        g_0:=[[starting_x + 1.5 * scaling, starting_y + 1 * scaling, starting_z + 20],[0,0,1,0],[0,0,0,0],[9E+09,9E+09,9E+09,9E+09,9E+09,9E+09]];
        g_1:=[[starting_x + 1.5 * scaling, starting_y + 1 * scaling, starting_z + 0],[0,0,1,0],[0,0,0,0],[9E+09,9E+09,9E+09,9E+09,9E+09,9E+09]];
        g_2:=[[starting_x + 0 * scaling, starting_y - 1 * scaling, starting_z + 0],[0,0,1,0],[0,0,0,0],[9E+09,9E+09,9E+09,9E+09,9E+09,9E+09]];
        g_3:=[[starting_x + 1 * scaling, starting_y - 3 * scaling, starting_z + 0],[0,0,1,0],[0,0,0,0],[9E+09,9E+09,9E+09,9E+09,9E+09,9E+09]];
        g_4:=[[starting_x + 3.5 * scaling, starting_y - 3.5 * scaling, starting_z + 0],[0,0,1,0],[0,0,0,0],[9E+09,9E+09,9E+09,9E+09,9E+09,9E+09]];
        g_5:=[[starting_x + 6 * scaling, starting_y - 2.5 * scaling, starting_z + 0],[0,0,1,0],[0,0,0,0],[9E+09,9E+09,9E+09,9E+09,9E+09,9E+09]];
        g_6:=[[starting_x + 7 * scaling, starting_y - 1 * scaling, starting_z + 0],[0,0,1,0],[0,0,0,0],[9E+09,9E+09,9E+09,9E+09,9E+09,9E+09]];
        g_7:=[[starting_x + 6 * scaling, starting_y + 1 * scaling, starting_z + 0],[0,0,1,0],[0,0,0,0],[9E+09,9E+09,9E+09,9E+09,9E+09,9E+09]];
        g_8:=[[starting_x + 1.5 * scaling, starting_y + 1 * scaling, starting_z + 0],[0,0,1,0],[0,0,0,0],[9E+09,9E+09,9E+09,9E+09,9E+09,9E+09]];
        g_9:=[[starting_x + 0 * scaling, starting_y + 2.5 * scaling, starting_z + 0],[0,0,1,0],[0,0,0,0],[9E+09,9E+09,9E+09,9E+09,9E+09,9E+09]];
        g_10:=[[starting_x + 1 * scaling, starting_y + 4 * scaling, starting_z + 0],[0,0,1,0],[0,0,0,0],[9E+09,9E+09,9E+09,9E+09,9E+09,9E+09]];
        g_11:=[[starting_x + 0 * scaling, starting_y + 6.5 * scaling, starting_z + 0],[0,0,1,0],[0,0,0,0],[9E+09,9E+09,9E+09,9E+09,9E+09,9E+09]];
        g_12:=[[starting_x + 3 * scaling, starting_y + 9 * scaling, starting_z + 0],[0,0,1,0],[0,0,0,0],[9E+09,9E+09,9E+09,9E+09,9E+09,9E+09]];
        g_13:=[[starting_x + 7.5 * scaling, starting_y + 9 * scaling, starting_z + 0],[0,0,1,0],[0,0,0,0],[9E+09,9E+09,9E+09,9E+09,9E+09,9E+09]];
        g_14:=[[starting_x + 4 * scaling, starting_y + 9 * scaling, starting_z + 0],[0,0,1,0],[0,0,0,0],[9E+09,9E+09,9E+09,9E+09,9E+09,9E+09]];
        g_15:=[[starting_x + 6 * scaling, starting_y + 7 * scaling, starting_z + 0],[0,0,1,0],[0,0,0,0],[9E+09,9E+09,9E+09,9E+09,9E+09,9E+09]];
        g_16:=[[starting_x + 6 * scaling, starting_y + 5 * scaling, starting_z + 0],[0,0,1,0],[0,0,0,0],[9E+09,9E+09,9E+09,9E+09,9E+09,9E+09]];
        g_17:=[[starting_x + 3.5 * scaling, starting_y + 3.5 * scaling, starting_z + 0],[0,0,1,0],[0,0,0,0],[9E+09,9E+09,9E+09,9E+09,9E+09,9E+09]];
        g_18:=[[starting_x + 1 * scaling, starting_y + 4 * scaling, starting_z + 0],[0,0,1,0],[0,0,0,0],[9E+09,9E+09,9E+09,9E+09,9E+09,9E+09]];
        g_19:=[[starting_x + 1 * scaling, starting_y + 4 * scaling, starting_z + 20],[0,0,1,0],[0,0,0,0],[9E+09,9E+09,9E+09,9E+09,9E+09,9E+09]];


        MoveL g_0,v50,fine,MyNewTool\WObj:=A3;
        MoveL g_1,v50,fine,MyNewTool\WObj:=A3;
	    MoveC g_2,g_3,v50,z1,MyNewTool\WObj:=A3;
        MoveC g_4,g_5,v50,z5,MyNewTool\WObj:=A3;
        MoveC g_6,g_7,v50,z5,MyNewTool\WObj:=A3;
        MoveL g_8,v50,fine,MyNewTool\WObj:=A3;
        MoveC g_9,g_10,v50,fine,MyNewTool\WObj:=A3;
        MoveC g_11,g_12,v50,fine,MyNewTool\WObj:=A3;
	    MoveL g_13,v50,fine,MyNewTool\WObj:=A3;
        MoveL g_14,v50,fine,MyNewTool\WObj:=A3;
        MoveC g_15,g_16,v50,z1,MyNewTool\WObj:=A3;
        MoveC g_17,g_18,v50,fine,MyNewTool\WObj:=A3;
        MoveL g_19,v50,fine,MyNewTool\WObj:=A3;


    ENDPROC


    PROC h(num starting_x, num starting_y, num starting_z, num scaling)
        VAR robtarget h_0;
        VAR robtarget h_1;
        VAR robtarget h_2;
	    VAR robtarget h_3;
	    VAR robtarget h_4;
	    VAR robtarget h_5;
	    VAR robtarget h_6;
        VAR robtarget h_7;
        VAR robtarget h_8;
        VAR robtarget h_9;

        h_0:=[[starting_x + 0 * scaling, starting_y + 0 * scaling, starting_z + 20],[0,0,1,0],[0,0,0,0],[9E+09,9E+09,9E+09,9E+09,9E+09,9E+09]];
        h_1:=[[starting_x + 0 * scaling, starting_y + 0 * scaling, starting_z + 0],[0,0,1,0],[0,0,0,0],[9E+09,9E+09,9E+09,9E+09,9E+09,9E+09]];
        h_2:=[[starting_x + 0 * scaling, starting_y + 14 * scaling, starting_z + 0],[0,0,1,0],[0,0,0,0],[9E+09,9E+09,9E+09,9E+09,9E+09,9E+09]];
        h_3:=[[starting_x + 0 * scaling, starting_y + 7 * scaling, starting_z + 0],[0,0,1,0],[0,0,0,0],[9E+09,9E+09,9E+09,9E+09,9E+09,9E+09]];
        h_4:=[[starting_x + 2 * scaling, starting_y + 8 * scaling, starting_z + 0],[0,0,1,0],[0,0,0,0],[9E+09,9E+09,9E+09,9E+09,9E+09,9E+09]];
        h_5:=[[starting_x + 4 * scaling, starting_y + 9 * scaling, starting_z + 0],[0,0,1,0],[0,0,0,0],[9E+09,9E+09,9E+09,9E+09,9E+09,9E+09]];
        h_6:=[[starting_x + 5.8 * scaling, starting_y + 7.2 * scaling, starting_z + 0],[0,0,1,0],[0,0,0,0],[9E+09,9E+09,9E+09,9E+09,9E+09,9E+09]];
        h_7:=[[starting_x + 6 * scaling, starting_y + 6 * scaling, starting_z + 0],[0,0,1,0],[0,0,0,0],[9E+09,9E+09,9E+09,9E+09,9E+09,9E+09]];
        h_8:=[[starting_x + 6 * scaling, starting_y + 0 * scaling, starting_z + 0],[0,0,1,0],[0,0,0,0],[9E+09,9E+09,9E+09,9E+09,9E+09,9E+09]];
        h_9:=[[starting_x + 6 * scaling, starting_y + 0 * scaling, starting_z + 20],[0,0,1,0],[0,0,0,0],[9E+09,9E+09,9E+09,9E+09,9E+09,9E+09]];

        MoveL h_0,v50,fine,MyNewTool\WObj:=A3;
        MoveL h_1,v50,fine,MyNewTool\WObj:=A3;
        MoveL h_2,v50,fine,MyNewTool\WObj:=A3;
        MoveL h_3,v50,fine,MyNewTool\WObj:=A3;
	    MoveL h_4,v50,fine,MyNewTool\WObj:=A3;
        MoveL h_5,v50,z5,MyNewTool\WObj:=A3;
        MoveC h_6,h_7,v50,fine,MyNewTool\WObj:=A3;
        MoveL h_8,v50,fine,MyNewTool\WObj:=A3;
        MoveL h_9,v50,fine,MyNewTool\WObj:=A3;

    ENDPROC

    PROC i(num starting_x, num starting_y, num starting_z, num scaling)
        VAR robtarget i_0;
        VAR robtarget i_1;
        VAR robtarget i_2;
	    VAR robtarget i_3;
	    VAR robtarget i_4;
	    VAR robtarget i_5;
	    VAR robtarget i_6;
        VAR robtarget i_7;


        i_0:=[[starting_x + 0 * scaling, starting_y + 0 * scaling, starting_z + 20],[0,0,1,0],[0,0,0,0],[9E+09,9E+09,9E+09,9E+09,9E+09,9E+09]];
        i_1:=[[starting_x + 0 * scaling, starting_y + 0 * scaling, starting_z + 0],[0,0,1,0],[0,0,0,0],[9E+09,9E+09,9E+09,9E+09,9E+09,9E+09]];
        i_2:=[[starting_x + 0 * scaling, starting_y + 9.5 * scaling, starting_z + 0],[0,0,1,0],[0,0,0,0],[9E+09,9E+09,9E+09,9E+09,9E+09,9E+09]];
        i_3:=[[starting_x + 0 * scaling, starting_y + 9.5 * scaling, starting_z + 20],[0,0,1,0],[0,0,0,0],[9E+09,9E+09,9E+09,9E+09,9E+09,9E+09]];
        i_4:=[[starting_x + 0 * scaling, starting_y + 12 * scaling, starting_z + 20],[0,0,1,0],[0,0,0,0],[9E+09,9E+09,9E+09,9E+09,9E+09,9E+09]];
        i_5:=[[starting_x + 0 * scaling, starting_y + 12 * scaling, starting_z + 0],[0,0,1,0],[0,0,0,0],[9E+09,9E+09,9E+09,9E+09,9E+09,9E+09]];
        i_6:=[[starting_x + 0 * scaling, starting_y + 12.1 * scaling, starting_z + 0],[0,0,1,0],[0,0,0,0],[9E+09,9E+09,9E+09,9E+09,9E+09,9E+09]];
        i_7:=[[starting_x + 0 * scaling, starting_y + 12.1 * scaling, starting_z + 20],[0,0,1,0],[0,0,0,0],[9E+09,9E+09,9E+09,9E+09,9E+09,9E+09]];


        MoveL i_0,v50,fine,MyNewTool\WObj:=A3;
        MoveL i_1,v50,fine,MyNewTool\WObj:=A3;
        MoveL i_2,v50,fine,MyNewTool\WObj:=A3;
        MoveL i_3,v50,fine,MyNewTool\WObj:=A3;
	    MoveL i_4,v50,fine,MyNewTool\WObj:=A3;
        MoveL i_5,v50,fine,MyNewTool\WObj:=A3;
        MoveL i_6,v50,fine,MyNewTool\WObj:=A3;
        MoveL i_7,v50,fine,MyNewTool\WObj:=A3;

    ENDPROC

    PROC j(num starting_x, num starting_y, num starting_z, num scaling)
        VAR robtarget j_0;
        VAR robtarget j_1;
        VAR robtarget j_2;
	    VAR robtarget j_3;
	    VAR robtarget j_4;
	    VAR robtarget j_5;
	    VAR robtarget j_6;
        VAR robtarget j_7;
        VAR robtarget j_8;
        VAR robtarget j_9;

        j_0:=[[starting_x - 1 * scaling, starting_y - 3 * scaling, starting_z + 20],[0,0,1,0],[0,0,0,0],[9E+09,9E+09,9E+09,9E+09,9E+09,9E+09]];
        j_1:=[[starting_x - 1 * scaling, starting_y - 3 * scaling, starting_z + 0],[0,0,1,0],[0,0,0,0],[9E+09,9E+09,9E+09,9E+09,9E+09,9E+09]];
        j_2:=[[starting_x + 1 * scaling, starting_y - 2.5 * scaling, starting_z + 0],[0,0,1,0],[0,0,0,0],[9E+09,9E+09,9E+09,9E+09,9E+09,9E+09]];
        j_3:=[[starting_x + 2 * scaling, starting_y - 1 * scaling, starting_z + 0],[0,0,1,0],[0,0,0,0],[9E+09,9E+09,9E+09,9E+09,9E+09,9E+09]];
        j_4:=[[starting_x + 2 * scaling, starting_y + 9.5 * scaling, starting_z + 0],[0,0,1,0],[0,0,0,0],[9E+09,9E+09,9E+09,9E+09,9E+09,9E+09]];
        j_5:=[[starting_x + 2 * scaling, starting_y + 9.5 * scaling, starting_z + 20],[0,0,1,0],[0,0,0,0],[9E+09,9E+09,9E+09,9E+09,9E+09,9E+09]];
        j_6:=[[starting_x + 2 * scaling, starting_y + 12 * scaling, starting_z + 20],[0,0,1,0],[0,0,0,0],[9E+09,9E+09,9E+09,9E+09,9E+09,9E+09]];
        j_7:=[[starting_x + 2 * scaling, starting_y + 12 * scaling, starting_z + 0],[0,0,1,0],[0,0,0,0],[9E+09,9E+09,9E+09,9E+09,9E+09,9E+09]];
        j_8:=[[starting_x + 2 * scaling, starting_y + 12.1 * scaling, starting_z + 0],[0,0,1,0],[0,0,0,0],[9E+09,9E+09,9E+09,9E+09,9E+09,9E+09]];
        j_9:=[[starting_x + 2 * scaling, starting_y + 12.1 * scaling, starting_z + 20],[0,0,1,0],[0,0,0,0],[9E+09,9E+09,9E+09,9E+09,9E+09,9E+09]];

        MoveL j_0,v50,fine,MyNewTool\WObj:=A3;
        MoveL j_1,v50,fine,MyNewTool\WObj:=A3;
        MoveC j_2,j_3,v50,z1,MyNewTool\WObj:=A3;
        MoveL j_4,v50,fine,MyNewTool\WObj:=A3;
	    MoveL j_5,v50,fine,MyNewTool\WObj:=A3;
        MoveL j_6,v50,fine,MyNewTool\WObj:=A3;
        MoveL j_7,v50,fine,MyNewTool\WObj:=A3;
        MoveL j_8,v50,fine,MyNewTool\WObj:=A3;
        MoveL j_9,v50,fine,MyNewTool\WObj:=A3;

    ENDPROC

    PROC k(num starting_x, num starting_y, num starting_z, num scaling)
        VAR robtarget k_0;
        VAR robtarget k_1;
        VAR robtarget k_2;
	    VAR robtarget k_3;
	    VAR robtarget k_4;
	    VAR robtarget k_5;
	    VAR robtarget k_6;
        VAR robtarget k_7;

        k_0:=[[starting_x + 0 * scaling, starting_y + 14 * scaling, starting_z + 20],[0,0,1,0],[0,0,0,0],[9E+09,9E+09,9E+09,9E+09,9E+09,9E+09]];
        k_1:=[[starting_x + 0 * scaling, starting_y + 14 * scaling, starting_z + 0],[0,0,1,0],[0,0,0,0],[9E+09,9E+09,9E+09,9E+09,9E+09,9E+09]];
        k_2:=[[starting_x + 0 * scaling, starting_y + 0 * scaling, starting_z + 0],[0,0,1,0],[0,0,0,0],[9E+09,9E+09,9E+09,9E+09,9E+09,9E+09]];
        k_3:=[[starting_x + 0 * scaling, starting_y + 5 * scaling, starting_z + 0],[0,0,1,0],[0,0,0,0],[9E+09,9E+09,9E+09,9E+09,9E+09,9E+09]];
        k_4:=[[starting_x + 5.8 * scaling, starting_y + 9 * scaling, starting_z + 0],[0,0,1,0],[0,0,0,0],[9E+09,9E+09,9E+09,9E+09,9E+09,9E+09]];
        k_5:=[[starting_x + 0 * scaling, starting_y + 5 * scaling, starting_z + 0],[0,0,1,0],[0,0,0,0],[9E+09,9E+09,9E+09,9E+09,9E+09,9E+09]];
        k_6:=[[starting_x + 6.2 * scaling, starting_y + 0 * scaling, starting_z + 0],[0,0,1,0],[0,0,0,0],[9E+09,9E+09,9E+09,9E+09,9E+09,9E+09]];
        k_7:=[[starting_x + 6.2 * scaling, starting_y + 0 * scaling, starting_z + 20],[0,0,1,0],[0,0,0,0],[9E+09,9E+09,9E+09,9E+09,9E+09,9E+09]];


        MoveL k_0,v50,fine,MyNewTool\WObj:=A3;
        MoveL k_1,v50,fine,MyNewTool\WObj:=A3;
        MoveL k_2,v50,fine,MyNewTool\WObj:=A3;
        MoveL k_3,v50,fine,MyNewTool\WObj:=A3;
	    MoveL k_4,v50,fine,MyNewTool\WObj:=A3;
        MoveL k_5,v50,z5,MyNewTool\WObj:=A3;
        MoveL k_6,v50,fine,MyNewTool\WObj:=A3;
        MoveL k_7,v50,fine,MyNewTool\WObj:=A3;

    ENDPROC
    PROC l(num starting_x, num starting_y, num starting_z, num scaling)
        VAR robtarget l_0;
        VAR robtarget l_1;
        VAR robtarget l_2;
        VAR robtarget l_3;


        l_0:=[[starting_x + 0 * scaling, starting_y + 0 * scaling, starting_z + 20],[0,0,1,0],[0,0,0,0],[9E+09,9E+09,9E+09,9E+09,9E+09,9E+09]];
        l_1:=[[starting_x + 0 * scaling, starting_y + 0 * scaling, starting_z + 0],[0,0,1,0],[0,0,0,0],[9E+09,9E+09,9E+09,9E+09,9E+09,9E+09]];
        l_2:=[[starting_x + 0 * scaling, starting_y + 14 * scaling, starting_z + 0],[0,0,1,0],[0,0,0,0],[9E+09,9E+09,9E+09,9E+09,9E+09,9E+09]];
        l_3:=[[starting_x + 0 * scaling, starting_y + 14 * scaling, starting_z + 20],[0,0,1,0],[0,0,0,0],[9E+09,9E+09,9E+09,9E+09,9E+09,9E+09]];


        MoveL l_0,v50,fine,MyNewTool\WObj:=A3;
        MoveL l_1,v50,fine,MyNewTool\WObj:=A3;
        MoveL l_2,v50,fine,MyNewTool\WObj:=A3;
        MoveL l_3,v50,fine,MyNewTool\WObj:=A3;

    ENDPROC

    PROC m(num starting_x, num starting_y, num starting_z, num scaling)
        VAR robtarget m_0;
        VAR robtarget m_1;
        VAR robtarget m_2;
        VAR robtarget m_3;
        VAR robtarget m_4;
        VAR robtarget m_5;
        VAR robtarget m_6;
        VAR robtarget m_7;
        VAR robtarget m_8;
        VAR robtarget m_9;
        VAR robtarget m_10;
        VAR robtarget m_11;
        VAR robtarget m_12;
        VAR robtarget m_13;


        m_0:=[[starting_x + 0 * scaling, starting_y + 0 * scaling, starting_z + 20],[0,0,1,0],[0,0,0,0],[9E+09,9E+09,9E+09,9E+09,9E+09,9E+09]];
        m_1:=[[starting_x + 0 * scaling, starting_y + 0 * scaling, starting_z + 0],[0,0,1,0],[0,0,0,0],[9E+09,9E+09,9E+09,9E+09,9E+09,9E+09]];
        m_2:=[[starting_x + 0 * scaling, starting_y + 9.5 * scaling, starting_z + 0],[0,0,1,0],[0,0,0,0],[9E+09,9E+09,9E+09,9E+09,9E+09,9E+09]];
        m_3:=[[starting_x + 0 * scaling, starting_y + 7 * scaling, starting_z + 0],[0,0,1,0],[0,0,0,0],[9E+09,9E+09,9E+09,9E+09,9E+09,9E+09]];
        m_4:=[[starting_x + 2 * scaling, starting_y + 8.5 * scaling, starting_z + 0],[0,0,1,0],[0,0,0,0],[9E+09,9E+09,9E+09,9E+09,9E+09,9E+09]];
        m_5:=[[starting_x + 4 * scaling, starting_y + 9 * scaling, starting_z + 0],[0,0,1,0],[0,0,0,0],[9E+09,9E+09,9E+09,9E+09,9E+09,9E+09]];
        m_6:=[[starting_x + 6 * scaling, starting_y + 8 * scaling, starting_z + 0],[0,0,1,0],[0,0,0,0],[9E+09,9E+09,9E+09,9E+09,9E+09,9E+09]];
        m_7:=[[starting_x + 6 * scaling, starting_y + 0 * scaling, starting_z + 0],[0,0,1,0],[0,0,0,0],[9E+09,9E+09,9E+09,9E+09,9E+09,9E+09]];
        m_8:=[[starting_x + 6 * scaling, starting_y + 7 * scaling, starting_z + 0],[0,0,1,0],[0,0,0,0],[9E+09,9E+09,9E+09,9E+09,9E+09,9E+09]];
        m_9:=[[starting_x + 7.4 * scaling, starting_y + 8.6 * scaling, starting_z + 0],[0,0,1,0],[0,0,0,0],[9E+09,9E+09,9E+09,9E+09,9E+09,9E+09]];
        m_10:=[[starting_x + 10 * scaling, starting_y + 9 * scaling, starting_z + 0],[0,0,1,0],[0,0,0,0],[9E+09,9E+09,9E+09,9E+09,9E+09,9E+09]];
        m_11:=[[starting_x + 12 * scaling, starting_y + 8 * scaling, starting_z + 0],[0,0,1,0],[0,0,0,0],[9E+09,9E+09,9E+09,9E+09,9E+09,9E+09]];
        m_12:=[[starting_x + 12 * scaling, starting_y + 0 * scaling, starting_z + 0],[0,0,1,0],[0,0,0,0],[9E+09,9E+09,9E+09,9E+09,9E+09,9E+09]];
        m_13:=[[starting_x + 12 * scaling, starting_y + 0 * scaling, starting_z + 20],[0,0,1,0],[0,0,0,0],[9E+09,9E+09,9E+09,9E+09,9E+09,9E+09]];

        MoveL m_0,v50,fine,MyNewTool\WObj:=A3;
        MoveL m_1,v50,fine,MyNewTool\WObj:=A3;
        MoveL m_2,v50,fine,MyNewTool\WObj:=A3;
        MoveL m_3,v50,fine,MyNewTool\WObj:=A3;
        MoveL m_4,v50,fine,MyNewTool\WObj:=A3;
        MoveC m_5,m_6,v50,z5,MyNewTool\WObj:=A3;
        MoveL m_7,v50,fine,MyNewTool\WObj:=A3;
        MoveL m_8,v50,fine,MyNewTool\WObj:=A3;
        MoveL m_9,v50,fine,MyNewTool\WObj:=A3;
        MoveC m_10,m_11,v50,z1,MyNewTool\WObj:=A3;
        MoveL m_12,v50,fine,MyNewTool\WObj:=A3;
        MoveL m_13,v50,fine,MyNewTool\WObj:=A3;

    ENDPROC

    PROC n(num starting_x, num starting_y, num starting_z, num scaling)
        VAR robtarget n_0;
        VAR robtarget n_1;
        VAR robtarget n_2;
        VAR robtarget n_3;
        VAR robtarget n_4;
        VAR robtarget n_5;
        VAR robtarget n_6;
        VAR robtarget n_7;
        VAR robtarget n_8;



        n_0:=[[starting_x + 0 * scaling, starting_y + 0 * scaling, starting_z + 20],[0,0,1,0],[0,0,0,0],[9E+09,9E+09,9E+09,9E+09,9E+09,9E+09]];
        n_1:=[[starting_x + 0 * scaling, starting_y + 0 * scaling, starting_z + 0],[0,0,1,0],[0,0,0,0],[9E+09,9E+09,9E+09,9E+09,9E+09,9E+09]];
        n_2:=[[starting_x + 0 * scaling, starting_y + 9.5 * scaling, starting_z + 0],[0,0,1,0],[0,0,0,0],[9E+09,9E+09,9E+09,9E+09,9E+09,9E+09]];
        n_3:=[[starting_x + 0 * scaling, starting_y + 7 * scaling, starting_z + 0],[0,0,1,0],[0,0,0,0],[9E+09,9E+09,9E+09,9E+09,9E+09,9E+09]];
        n_4:=[[starting_x + 2 * scaling, starting_y + 8.5 * scaling, starting_z + 0],[0,0,1,0],[0,0,0,0],[9E+09,9E+09,9E+09,9E+09,9E+09,9E+09]];
        n_5:=[[starting_x + 4 * scaling, starting_y + 9 * scaling, starting_z + 0],[0,0,1,0],[0,0,0,0],[9E+09,9E+09,9E+09,9E+09,9E+09,9E+09]];
        n_6:=[[starting_x + 6 * scaling, starting_y + 8 * scaling, starting_z + 0],[0,0,1,0],[0,0,0,0],[9E+09,9E+09,9E+09,9E+09,9E+09,9E+09]];
        n_7:=[[starting_x + 6 * scaling, starting_y + 0 * scaling, starting_z + 0],[0,0,1,0],[0,0,0,0],[9E+09,9E+09,9E+09,9E+09,9E+09,9E+09]];
        n_8:=[[starting_x + 6 * scaling, starting_y + 0 * scaling, starting_z + 20],[0,0,1,0],[0,0,0,0],[9E+09,9E+09,9E+09,9E+09,9E+09,9E+09]];


        MoveL n_0,v50,fine,MyNewTool\WObj:=A3;
        MoveL n_1,v50,fine,MyNewTool\WObj:=A3;
        MoveL n_2,v50,fine,MyNewTool\WObj:=A3;
        MoveL n_3,v50,fine,MyNewTool\WObj:=A3;
        MoveL n_4,v50,fine,MyNewTool\WObj:=A3;
        MoveC n_5,n_6,v50,z5,MyNewTool\WObj:=A3;
        MoveL n_7,v50,fine,MyNewTool\WObj:=A3;
        MoveL n_8,v50,fine,MyNewTool\WObj:=A3;


    ENDPROC

    PROC o(num starting_x, num starting_y, num starting_z, num scaling)
        VAR robtarget o_0;
        VAR robtarget o_1;
        VAR robtarget o_2;
        VAR robtarget o_3;
        VAR robtarget o_4;
        VAR robtarget o_5;
        VAR robtarget o_6;


        o_0:=[[starting_x + 2 * scaling, starting_y + 0.5 * scaling, starting_z + 20],[0,0,1,0],[0,0,0,0],[9E+09,9E+09,9E+09,9E+09,9E+09,9E+09]];
        o_1:=[[starting_x + 2 * scaling, starting_y + 0.5 * scaling, starting_z + 0],[0,0,1,0],[0,0,0,0],[9E+09,9E+09,9E+09,9E+09,9E+09,9E+09]];
        o_2:=[[starting_x + 2 * scaling, starting_y + 7 * scaling, starting_z + 0],[0,0,1,0],[0,0,0,0],[9E+09,9E+09,9E+09,9E+09,9E+09,9E+09]];
        o_3:=[[starting_x + 5.5 * scaling, starting_y + 7 * scaling, starting_z + 0],[0,0,1,0],[0,0,0,0],[9E+09,9E+09,9E+09,9E+09,9E+09,9E+09]];
        o_4:=[[starting_x + 5.5 * scaling, starting_y + 0.5 * scaling, starting_z + 0],[0,0,1,0],[0,0,0,0],[9E+09,9E+09,9E+09,9E+09,9E+09,9E+09]];
        o_5:=[[starting_x + 2 * scaling, starting_y + 0.5 * scaling, starting_z + 0],[0,0,1,0],[0,0,0,0],[9E+09,9E+09,9E+09,9E+09,9E+09,9E+09]];
        o_6:=[[starting_x + 2 * scaling, starting_y + 0.5 * scaling, starting_z + 20],[0,0,1,0],[0,0,0,0],[9E+09,9E+09,9E+09,9E+09,9E+09,9E+09]];

        MoveL o_0,v50,fine,MyNewTool\WObj:=A3;
        MoveL o_1,v50,fine,MyNewTool\WObj:=A3;
        MoveC o_2,o_3,v50,fine,MyNewTool\WObj:=A3;
        MoveC o_4,o_5,v50,fine,MyNewTool\WObj:=A3;
        MoveL o_6,v50,fine,MyNewTool\WObj:=A3;

    ENDPROC

    PROC p(num starting_x, num starting_y, num starting_z, num scaling)
        VAR robtarget p_0;
        VAR robtarget p_1;
        VAR robtarget p_2;
	    VAR robtarget p_3;
	    VAR robtarget p_4;
	    VAR robtarget p_5;
	    VAR robtarget p_6;
	    VAR robtarget p_7;
	    VAR robtarget p_8;
	    VAR robtarget p_9;
	    VAR robtarget p_10;

        p_0:=[[starting_x + 0* scaling, starting_y - 3.5 * scaling, starting_z + 20],[0,0,1,0],[0,0,0,0],[9E+09,9E+09,9E+09,9E+09,9E+09,9E+09]];
        p_1:=[[starting_x + 0 * scaling, starting_y - 3.5 * scaling, starting_z + 0],[0,0,1,0],[0,0,0,0],[9E+09,9E+09,9E+09,9E+09,9E+09,9E+09]];
        p_2:=[[starting_x + 0 * scaling, starting_y + 9 * scaling, starting_z + 0],[0,0,1,0],[0,0,0,0],[9E+09,9E+09,9E+09,9E+09,9E+09,9E+09]];
        p_3:=[[starting_x + 0 * scaling, starting_y + 7 * scaling, starting_z + 0],[0,0,1,0],[0,0,0,0],[9E+09,9E+09,9E+09,9E+09,9E+09,9E+09]];
        p_4:=[[starting_x + 3 * scaling, starting_y + 9 * scaling, starting_z + 0],[0,0,1,0],[0,0,0,0],[9E+09,9E+09,9E+09,9E+09,9E+09,9E+09]];
        p_5:=[[starting_x + 6 * scaling, starting_y + 8 * scaling, starting_z + 0],[0,0,1,0],[0,0,0,0],[9E+09,9E+09,9E+09,9E+09,9E+09,9E+09]];
        p_6:=[[starting_x + 7 * scaling, starting_y + 4.5 * scaling, starting_z + 0],[0,0,1,0],[0,0,0,0],[9E+09,9E+09,9E+09,9E+09,9E+09,9E+09]];
        p_7:=[[starting_x + 6 * scaling, starting_y + 1 * scaling, starting_z + 0],[0,0,1,0],[0,0,0,0],[9E+09,9E+09,9E+09,9E+09,9E+09,9E+09]];
        p_8:=[[starting_x + 4 * scaling, starting_y + 0 * scaling, starting_z + 0],[0,0,1,0],[0,0,0,0],[9E+09,9E+09,9E+09,9E+09,9E+09,9E+09]];
        p_9:=[[starting_x + 0 * scaling, starting_y + 2 * scaling, starting_z + 0],[0,0,1,0],[0,0,0,0],[9E+09,9E+09,9E+09,9E+09,9E+09,9E+09]];
        p_10:=[[starting_x + 0 * scaling, starting_y + 2 * scaling, starting_z + 20],[0,0,1,0],[0,0,0,0],[9E+09,9E+09,9E+09,9E+09,9E+09,9E+09]];

        MoveL p_0,v50,fine,MyNewTool\WObj:=A3;
	    MoveL p_1,v50,fine,MyNewTool\WObj:=A3;
        MoveL p_2,v50,fine,MyNewTool\WObj:=A3;
        MoveL p_3,v50,fine,MyNewTool\WObj:=A3;
	    MoveC p_4,p_5,v50,z1,MyNewTool\WObj:=A3;
	    MoveC p_6,p_7,v50,z1,MyNewTool\WObj:=A3;
	    MoveC p_8,p_9,v50,fine,MyNewTool\WObj:=A3;
	    MoveL p_10,v50,fine,MyNewTool\WObj:=A3;

	ENDPROC

    PROC q(num starting_x, num starting_y, num starting_z, num scaling)
        VAR robtarget q_0;
        VAR robtarget q_1;
        VAR robtarget q_2;
	    VAR robtarget q_3;
	    VAR robtarget q_4;
	    VAR robtarget q_5;
	    VAR robtarget q_6;
	    VAR robtarget q_7;
	    VAR robtarget q_8;
	    VAR robtarget q_9;
	    VAR robtarget q_10;

        q_0:=[[starting_x + 7 * scaling, starting_y - 4 * scaling, starting_z + 20],[0,0,1,0],[0,0,0,0],[9E+09,9E+09,9E+09,9E+09,9E+09,9E+09]];
        q_1:=[[starting_x + 7 * scaling, starting_y -4 * scaling, starting_z + 0],[0,0,1,0],[0,0,0,0],[9E+09,9E+09,9E+09,9E+09,9E+09,9E+09]];
        q_2:=[[starting_x + 7 * scaling, starting_y + 9 * scaling, starting_z + 0],[0,0,1,0],[0,0,0,0],[9E+09,9E+09,9E+09,9E+09,9E+09,9E+09]];
        q_3:=[[starting_x + 7 * scaling, starting_y + 7 * scaling, starting_z + 0],[0,0,1,0],[0,0,0,0],[9E+09,9E+09,9E+09,9E+09,9E+09,9E+09]];
        q_4:=[[starting_x + 4 * scaling, starting_y + 9 * scaling, starting_z + 0],[0,0,1,0],[0,0,0,0],[9E+09,9E+09,9E+09,9E+09,9E+09,9E+09]];
        q_5:=[[starting_x + 1 * scaling, starting_y + 8 * scaling, starting_z + 0],[0,0,1,0],[0,0,0,0],[9E+09,9E+09,9E+09,9E+09,9E+09,9E+09]];
        q_6:=[[starting_x + 0 * scaling, starting_y + 4.5 * scaling, starting_z + 0],[0,0,1,0],[0,0,0,0],[9E+09,9E+09,9E+09,9E+09,9E+09,9E+09]];
        q_7:=[[starting_x + 1 * scaling, starting_y + 1 * scaling, starting_z + 0],[0,0,1,0],[0,0,0,0],[9E+09,9E+09,9E+09,9E+09,9E+09,9E+09]];
        q_8:=[[starting_x + 3 * scaling, starting_y + 0 * scaling, starting_z + 0],[0,0,1,0],[0,0,0,0],[9E+09,9E+09,9E+09,9E+09,9E+09,9E+09]];
        q_9:=[[starting_x + 7 * scaling, starting_y + 2 * scaling, starting_z + 0],[0,0,1,0],[0,0,0,0],[9E+09,9E+09,9E+09,9E+09,9E+09,9E+09]];
        q_10:=[[starting_x + 7 * scaling, starting_y + 2 * scaling, starting_z + 20],[0,0,1,0],[0,0,0,0],[9E+09,9E+09,9E+09,9E+09,9E+09,9E+09]];

        MoveL q_0,v50,fine,MyNewTool\WObj:=A3;
	    MoveL q_1,v50,fine,MyNewTool\WObj:=A3;
        MoveL q_2,v50,fine,MyNewTool\WObj:=A3;
        MoveL q_3,v50,fine,MyNewTool\WObj:=A3;
	    MoveC q_4,q_5,v50,z1,MyNewTool\WObj:=A3;
	    MoveC q_6,q_7,v50,z1,MyNewTool\WObj:=A3;
	    MoveC q_8,q_9,v50,fine,MyNewTool\WObj:=A3;
	    MoveL q_10,v50,fine,MyNewTool\WObj:=A3;

	ENDPROC

    PROC r(num starting_x, num starting_y, num starting_z, num scaling)
        VAR robtarget r_0;
        VAR robtarget r_1;
        VAR robtarget r_2;
        VAR robtarget r_3;
        VAR robtarget r_4;
        VAR robtarget r_5;
        VAR robtarget r_6;
        VAR robtarget r_7;
        VAR robtarget r_8;



        r_0:=[[starting_x + 0 * scaling, starting_y + 0 * scaling, starting_z + 20],[0,0,1,0],[0,0,0,0],[9E+09,9E+09,9E+09,9E+09,9E+09,9E+09]];
        r_1:=[[starting_x + 0 * scaling, starting_y + 0 * scaling, starting_z + 0],[0,0,1,0],[0,0,0,0],[9E+09,9E+09,9E+09,9E+09,9E+09,9E+09]];
        r_2:=[[starting_x + 0 * scaling, starting_y + 9.5 * scaling, starting_z + 0],[0,0,1,0],[0,0,0,0],[9E+09,9E+09,9E+09,9E+09,9E+09,9E+09]];
        r_3:=[[starting_x + 0 * scaling, starting_y + 7 * scaling, starting_z + 0],[0,0,1,0],[0,0,0,0],[9E+09,9E+09,9E+09,9E+09,9E+09,9E+09]];
        r_4:=[[starting_x + 2 * scaling, starting_y + 8.5 * scaling, starting_z + 0],[0,0,1,0],[0,0,0,0],[9E+09,9E+09,9E+09,9E+09,9E+09,9E+09]];
        r_5:=[[starting_x + 4 * scaling, starting_y + 9 * scaling, starting_z + 0],[0,0,1,0],[0,0,0,0],[9E+09,9E+09,9E+09,9E+09,9E+09,9E+09]];
        r_6:=[[starting_x + 6 * scaling, starting_y + 8 * scaling, starting_z + 0],[0,0,1,0],[0,0,0,0],[9E+09,9E+09,9E+09,9E+09,9E+09,9E+09]];
        r_7:=[[starting_x + 6 * scaling, starting_y + 8 * scaling, starting_z + 20],[0,0,1,0],[0,0,0,0],[9E+09,9E+09,9E+09,9E+09,9E+09,9E+09]];



        MoveL r_0,v50,fine,MyNewTool\WObj:=A3;
        MoveL r_1,v50,fine,MyNewTool\WObj:=A3;
        MoveL r_2,v50,fine,MyNewTool\WObj:=A3;
        MoveL r_3,v50,fine,MyNewTool\WObj:=A3;
        MoveL r_4,v50,fine,MyNewTool\WObj:=A3;
        MoveC r_5,r_6,v50,fine,MyNewTool\WObj:=A3;
        MoveL r_7,v50,fine,MyNewTool\WObj:=A3;

    ENDPROC

    PROC s(num starting_x, num starting_y, num starting_z, num scaling)
        VAR robtarget s_0;
        VAR robtarget s_1;
        VAR robtarget s_2;
	    VAR robtarget s_3;
	    VAR robtarget s_4;
	    VAR robtarget s_5;
	    VAR robtarget s_6;
        VAR robtarget s_7;
        VAR robtarget s_8;
        VAR robtarget s_9;
        VAR robtarget s_10;
        VAR robtarget s_11;

        s_0:=[[starting_x + 0 * scaling, starting_y + 2 * scaling, starting_z + 20],[0,0,1,0],[0,0,0,0],[9E+09,9E+09,9E+09,9E+09,9E+09,9E+09]];
        s_1:=[[starting_x + 0 * scaling, starting_y + 2 * scaling, starting_z + 0],[0,0,1,0],[0,0,0,0],[9E+09,9E+09,9E+09,9E+09,9E+09,9E+09]];
        s_2:=[[starting_x + 2.5 * scaling, starting_y + 0 * scaling, starting_z + 0],[0,0,1,0],[0,0,0,0],[9E+09,9E+09,9E+09,9E+09,9E+09,9E+09]];
        s_3:=[[starting_x + 5 * scaling, starting_y + 1 * scaling, starting_z + 0],[0,0,1,0],[0,0,0,0],[9E+09,9E+09,9E+09,9E+09,9E+09,9E+09]];
        s_4:=[[starting_x + 5.5 * scaling, starting_y + 2 * scaling, starting_z + 0],[0,0,1,0],[0,0,0,0],[9E+09,9E+09,9E+09,9E+09,9E+09,9E+09]];
        s_5:=[[starting_x + 4 * scaling, starting_y + 4 * scaling, starting_z + 0],[0,0,1,0],[0,0,0,0],[9E+09,9E+09,9E+09,9E+09,9E+09,9E+09]];
        s_6:=[[starting_x + 1 * scaling, starting_y + 6 * scaling, starting_z + 0],[0,0,1,0],[0,0,0,0],[9E+09,9E+09,9E+09,9E+09,9E+09,9E+09]];
        s_7:=[[starting_x + 0.5 * scaling, starting_y + 7.5 * scaling, starting_z + 0],[0,0,1,0],[0,0,0,0],[9E+09,9E+09,9E+09,9E+09,9E+09,9E+09]];
        s_8:=[[starting_x + 1 * scaling, starting_y + 9 * scaling, starting_z + 0],[0,0,1,0],[0,0,0,0],[9E+09,9E+09,9E+09,9E+09,9E+09,9E+09]];
        s_9:=[[starting_x + 4 * scaling, starting_y + 9.5 * scaling, starting_z + 0],[0,0,1,0],[0,0,0,0],[9E+09,9E+09,9E+09,9E+09,9E+09,9E+09]];
        s_10:=[[starting_x + 5.5 * scaling, starting_y + 8 * scaling, starting_z + 0],[0,0,1,0],[0,0,0,0],[9E+09,9E+09,9E+09,9E+09,9E+09,9E+09]];
        s_11:=[[starting_x + 5.5 * scaling, starting_y + 8 * scaling, starting_z + 20],[0,0,1,0],[0,0,0,0],[9E+09,9E+09,9E+09,9E+09,9E+09,9E+09]];

        MoveL s_0,v50,fine,MyNewTool\WObj:=A3;
        MoveL s_1,v50,fine,MyNewTool\WObj:=A3;
        MoveC s_2,s_3,v50,z5,MyNewTool\WObj:=A3;
        MoveC s_4,s_5,v50,z5,MyNewTool\WObj:=A3;
        MoveL s_6,v50,z5,MyNewTool\WObj:=A3;
        MoveC s_7,s_8,v50,z5,MyNewTool\WObj:=A3;
        MoveC s_9,s_10,v50,fine,MyNewTool\WObj:=A3;
        MoveL s_11,v50,fine,MyNewTool\WObj:=A3;

    ENDPROC
    PROC t(num starting_x, num starting_y, num starting_z, num scaling)
        VAR robtarget t_0;
        VAR robtarget t_1;
        VAR robtarget t_2;
	    VAR robtarget t_3;
	    VAR robtarget t_4;
	    VAR robtarget t_5;
	    VAR robtarget t_6;
        VAR robtarget t_7;
        VAR robtarget t_8;
        VAR robtarget t_9;

        t_0:=[[starting_x + 2 * scaling, starting_y + 12 * scaling, starting_z + 20],[0,0,1,0],[0,0,0,0],[9E+09,9E+09,9E+09,9E+09,9E+09,9E+09]];
        t_1:=[[starting_x + 2 * scaling, starting_y + 12 * scaling, starting_z + 0],[0,0,1,0],[0,0,0,0],[9E+09,9E+09,9E+09,9E+09,9E+09,9E+09]];
        t_2:=[[starting_x + 2 * scaling, starting_y + 2 * scaling, starting_z + 0],[0,0,1,0],[0,0,0,0],[9E+09,9E+09,9E+09,9E+09,9E+09,9E+09]];
        t_3:=[[starting_x + 3 * scaling, starting_y + 0.5 * scaling, starting_z + 0],[0,0,1,0],[0,0,0,0],[9E+09,9E+09,9E+09,9E+09,9E+09,9E+09]];
        t_4:=[[starting_x + 5.5 * scaling, starting_y + 1 * scaling, starting_z + 0],[0,0,1,0],[0,0,0,0],[9E+09,9E+09,9E+09,9E+09,9E+09,9E+09]];
        t_5:=[[starting_x + 5.5 * scaling, starting_y + 1 * scaling, starting_z + 20],[0,0,1,0],[0,0,0,0],[9E+09,9E+09,9E+09,9E+09,9E+09,9E+09]];
        t_6:=[[starting_x + 0 * scaling, starting_y + 9 * scaling, starting_z + 20],[0,0,1,0],[0,0,0,0],[9E+09,9E+09,9E+09,9E+09,9E+09,9E+09]];
        t_7:=[[starting_x + 0 * scaling, starting_y + 9 * scaling, starting_z + 0],[0,0,1,0],[0,0,0,0],[9E+09,9E+09,9E+09,9E+09,9E+09,9E+09]];
        t_8:=[[starting_x + 5 * scaling, starting_y + 9 * scaling, starting_z + 0],[0,0,1,0],[0,0,0,0],[9E+09,9E+09,9E+09,9E+09,9E+09,9E+09]];
        t_9:=[[starting_x + 5 * scaling, starting_y + 9 * scaling, starting_z + 20],[0,0,1,0],[0,0,0,0],[9E+09,9E+09,9E+09,9E+09,9E+09,9E+09]];

        MoveL t_0,v50,fine,MyNewTool\WObj:=A3;
        MoveL t_1,v50,fine,MyNewTool\WObj:=A3;
        MoveL t_2,v50,fine,MyNewTool\WObj:=A3;
	    MoveC t_3,t_4,v50,fine,MyNewTool\WObj:=A3;
        MoveL t_5,v50,fine,MyNewTool\WObj:=A3;
	    MoveL t_6,v50,fine,MyNewTool\WObj:=A3;
        MoveL t_7,v50,fine,MyNewTool\WObj:=A3;
        MoveL t_8,v50,fine,MyNewTool\WObj:=A3;
        MoveL t_9,v50,fine,MyNewTool\WObj:=A3;

    ENDPROC

    PROC u(num starting_x, num starting_y, num starting_z, num scaling)
        VAR robtarget u_0;
        VAR robtarget u_1;
        VAR robtarget u_2;
        VAR robtarget u_3;
        VAR robtarget u_4;
        VAR robtarget u_5;
        VAR robtarget u_6;
        VAR robtarget u_7;
        VAR robtarget u_8;

        u_0:=[[starting_x + 6 * scaling, starting_y + 9.5 * scaling, starting_z + 20],[0,0,1,0],[0,0,0,0],[9E+09,9E+09,9E+09,9E+09,9E+09,9E+09]];
        u_1:=[[starting_x + 6 * scaling, starting_y + 9.5 * scaling, starting_z + 0],[0,0,1,0],[0,0,0,0],[9E+09,9E+09,9E+09,9E+09,9E+09,9E+09]];
        u_2:=[[starting_x + 6 * scaling, starting_y + 0 * scaling, starting_z + 0],[0,0,1,0],[0,0,0,0],[9E+09,9E+09,9E+09,9E+09,9E+09,9E+09]];
        u_3:=[[starting_x + 6 * scaling, starting_y + 2 * scaling, starting_z + 0],[0,0,1,0],[0,0,0,0],[9E+09,9E+09,9E+09,9E+09,9E+09,9E+09]];
        u_4:=[[starting_x + 4 * scaling, starting_y + 1 * scaling, starting_z + 0],[0,0,1,0],[0,0,0,0],[9E+09,9E+09,9E+09,9E+09,9E+09,9E+09]];
        u_5:=[[starting_x + 2 * scaling, starting_y + 0.5 * scaling, starting_z + 0],[0,0,1,0],[0,0,0,0],[9E+09,9E+09,9E+09,9E+09,9E+09,9E+09]];
        u_6:=[[starting_x + 0 * scaling, starting_y + 1.5 * scaling, starting_z + 0],[0,0,1,0],[0,0,0,0],[9E+09,9E+09,9E+09,9E+09,9E+09,9E+09]];
        u_7:=[[starting_x + 0 * scaling, starting_y + 9.5 * scaling, starting_z + 0],[0,0,1,0],[0,0,0,0],[9E+09,9E+09,9E+09,9E+09,9E+09,9E+09]];
        u_8:=[[starting_x + 0 * scaling, starting_y + 9.5 * scaling, starting_z + 20],[0,0,1,0],[0,0,0,0],[9E+09,9E+09,9E+09,9E+09,9E+09,9E+09]];

        MoveL u_0,v50,fine,MyNewTool\WObj:=A3;
        MoveL u_1,v50,fine,MyNewTool\WObj:=A3;
        MoveL u_2,v50,fine,MyNewTool\WObj:=A3;
        MoveL u_3,v50,fine,MyNewTool\WObj:=A3;
        MoveL u_4,v50,fine,MyNewTool\WObj:=A3;
        MoveC u_5,u_6,v50,z5,MyNewTool\WObj:=A3;
        MoveL u_7,v50,fine,MyNewTool\WObj:=A3;
        MoveL u_8,v50,fine,MyNewTool\WObj:=A3;

    ENDPROC

    PROC v(num starting_x, num starting_y, num starting_z, num scaling)
        VAR robtarget v_0;
        VAR robtarget v_1;
        VAR robtarget v_2;
        VAR robtarget v_3;
        VAR robtarget v_4;

        v_0:=[[starting_x + 0 * scaling, starting_y + 9 * scaling, starting_z + 20],[0,0,1,0],[0,0,0,0],[9E+09,9E+09,9E+09,9E+09,9E+09,9E+09]];
        v_1:=[[starting_x + 0 * scaling, starting_y + 9 * scaling, starting_z + 0],[0,0,1,0],[0,0,0,0],[9E+09,9E+09,9E+09,9E+09,9E+09,9E+09]];
        v_2:=[[starting_x + 4 * scaling, starting_y + 0 * scaling, starting_z + 0],[0,0,1,0],[0,0,0,0],[9E+09,9E+09,9E+09,9E+09,9E+09,9E+09]];
        v_3:=[[starting_x + 8 * scaling, starting_y + 9 * scaling, starting_z + 0],[0,0,1,0],[0,0,0,0],[9E+09,9E+09,9E+09,9E+09,9E+09,9E+09]];
        v_4:=[[starting_x + 8 * scaling, starting_y + 9 * scaling, starting_z + 20],[0,0,1,0],[0,0,0,0],[9E+09,9E+09,9E+09,9E+09,9E+09,9E+09]];

        MoveL v_0,v50,fine,MyNewTool\WObj:=A3;
        MoveL v_1,v50,fine,MyNewTool\WObj:=A3;
        MoveL v_2,v50,fine,MyNewTool\WObj:=A3;
        MoveL v_3,v50,fine,MyNewTool\WObj:=A3;
        MoveL v_4,v50,fine,MyNewTool\WObj:=A3;

    ENDPROC

    PROC w(num starting_x, num starting_y, num starting_z, num scaling)
        VAR robtarget w_0;
        VAR robtarget w_1;
        VAR robtarget w_2;
        VAR robtarget w_3;
        VAR robtarget w_4;
        VAR robtarget w_5;
        VAR robtarget w_6;

        w_0:=[[starting_x + 0 * scaling, starting_y + 9 * scaling, starting_z + 20],[0,0,1,0],[0,0,0,0],[9E+09,9E+09,9E+09,9E+09,9E+09,9E+09]];
        w_1:=[[starting_x + 0 * scaling, starting_y + 9 * scaling, starting_z + 0],[0,0,1,0],[0,0,0,0],[9E+09,9E+09,9E+09,9E+09,9E+09,9E+09]];
        w_2:=[[starting_x + 3 * scaling, starting_y + 0 * scaling, starting_z + 0],[0,0,1,0],[0,0,0,0],[9E+09,9E+09,9E+09,9E+09,9E+09,9E+09]];
        w_3:=[[starting_x + 6 * scaling, starting_y + 9 * scaling, starting_z + 0],[0,0,1,0],[0,0,0,0],[9E+09,9E+09,9E+09,9E+09,9E+09,9E+09]];
        w_4:=[[starting_x + 9 * scaling, starting_y + 0 * scaling, starting_z + 0],[0,0,1,0],[0,0,0,0],[9E+09,9E+09,9E+09,9E+09,9E+09,9E+09]];
        w_5:=[[starting_x + 12 * scaling, starting_y + 9 * scaling, starting_z + 0],[0,0,1,0],[0,0,0,0],[9E+09,9E+09,9E+09,9E+09,9E+09,9E+09]];
        w_6:=[[starting_x + 12 * scaling, starting_y + 9 * scaling, starting_z + 20],[0,0,1,0],[0,0,0,0],[9E+09,9E+09,9E+09,9E+09,9E+09,9E+09]];


        MoveL w_0,v50,fine,MyNewTool\WObj:=A3;
        MoveL w_1,v50,fine,MyNewTool\WObj:=A3;
        MoveL w_2,v50,fine,MyNewTool\WObj:=A3;
        MoveL w_3,v50,fine,MyNewTool\WObj:=A3;
        MoveL w_4,v50,fine,MyNewTool\WObj:=A3;
        MoveL w_5,v50,fine,MyNewTool\WObj:=A3;
        MoveL w_6,v50,fine,MyNewTool\WObj:=A3;

    ENDPROC

    PROC x_draw(num starting_x, num starting_y, num starting_z, num scaling)
        VAR robtarget x_0;
        VAR robtarget x_1;
        VAR robtarget x_2;
        VAR robtarget x_3;
        VAR robtarget x_4;
        VAR robtarget x_5;
        VAR robtarget x_6;
        VAR robtarget x_7;

        x_0:=[[starting_x + 0 * scaling, starting_y + 0 * scaling, starting_z + 20],[0,0,1,0],[0,0,0,0],[9E+09,9E+09,9E+09,9E+09,9E+09,9E+09]];
        x_1:=[[starting_x + 0 * scaling, starting_y + 0 * scaling, starting_z + 0],[0,0,1,0],[0,0,0,0],[9E+09,9E+09,9E+09,9E+09,9E+09,9E+09]];
        x_2:=[[starting_x + 6 * scaling, starting_y + 9 * scaling, starting_z + 0],[0,0,1,0],[0,0,0,0],[9E+09,9E+09,9E+09,9E+09,9E+09,9E+09]];
        x_3:=[[starting_x + 6 * scaling, starting_y + 9 * scaling, starting_z + 20],[0,0,1,0],[0,0,0,0],[9E+09,9E+09,9E+09,9E+09,9E+09,9E+09]];
        x_4:=[[starting_x + 0 * scaling, starting_y + 9 * scaling, starting_z + 20],[0,0,1,0],[0,0,0,0],[9E+09,9E+09,9E+09,9E+09,9E+09,9E+09]];
        x_5:=[[starting_x + 0 * scaling, starting_y + 9 * scaling, starting_z + 0],[0,0,1,0],[0,0,0,0],[9E+09,9E+09,9E+09,9E+09,9E+09,9E+09]];
        x_6:=[[starting_x + 6 * scaling, starting_y + 0 * scaling, starting_z + 0],[0,0,1,0],[0,0,0,0],[9E+09,9E+09,9E+09,9E+09,9E+09,9E+09]];
        x_7:=[[starting_x + 6 * scaling, starting_y + 0 * scaling, starting_z + 20],[0,0,1,0],[0,0,0,0],[9E+09,9E+09,9E+09,9E+09,9E+09,9E+09]];

        MoveL x_0,v50,fine,MyNewTool\WObj:=A3;
        MoveL x_1,v50,fine,MyNewTool\WObj:=A3;
        MoveL x_2,v50,fine,MyNewTool\WObj:=A3;
        MoveL x_3,v50,fine,MyNewTool\WObj:=A3;
        MoveL x_4,v50,fine,MyNewTool\WObj:=A3;
        MoveL x_5,v50,fine,MyNewTool\WObj:=A3;
        MoveL x_6,v50,fine,MyNewTool\WObj:=A3;
        MoveL x_7,v50,fine,MyNewTool\WObj:=A3;

    ENDPROC

    PROC y_draw(num starting_x, num starting_y, num starting_z, num scaling)
        VAR robtarget y_0;
        VAR robtarget y_1;
        VAR robtarget y_2;
        VAR robtarget y_3;
        VAR robtarget y_4;
        VAR robtarget y_5;
        VAR robtarget y_6;
        VAR robtarget y_7;

        y_0:=[[starting_x + 6 * scaling, starting_y + 9 * scaling, starting_z + 20],[0,0,1,0],[0,0,0,0],[9E+09,9E+09,9E+09,9E+09,9E+09,9E+09]];
        y_1:=[[starting_x + 6 * scaling, starting_y + 9 * scaling, starting_z + 0],[0,0,1,0],[0,0,0,0],[9E+09,9E+09,9E+09,9E+09,9E+09,9E+09]];
        y_2:=[[starting_x + 2.5 * scaling, starting_y - 3 * scaling, starting_z + 0],[0,0,1,0],[0,0,0,0],[9E+09,9E+09,9E+09,9E+09,9E+09,9E+09]];
        y_3:=[[starting_x + 3.35 * scaling, starting_y + 0 * scaling, starting_z + 0],[0,0,1,0],[0,0,0,0],[9E+09,9E+09,9E+09,9E+09,9E+09,9E+09]];
        y_4:=[[starting_x + 0 * scaling, starting_y + 9 * scaling, starting_z + 0],[0,0,1,0],[0,0,0,0],[9E+09,9E+09,9E+09,9E+09,9E+09,9E+09]];
        y_5:=[[starting_x + 0 * scaling, starting_y + 9 * scaling, starting_z + 20],[0,0,1,0],[0,0,0,0],[9E+09,9E+09,9E+09,9E+09,9E+09,9E+09]];

        MoveL y_0,v50,fine,MyNewTool\WObj:=A3;
        MoveL y_1,v50,fine,MyNewTool\WObj:=A3;
        MoveL y_2,v50,fine,MyNewTool\WObj:=A3;
        MoveL y_3,v50,fine,MyNewTool\WObj:=A3;
        MoveL y_4,v50,fine,MyNewTool\WObj:=A3;
        MoveL y_5,v50,fine,MyNewTool\WObj:=A3;


    ENDPROC

    PROC z_draw(num starting_x, num starting_y, num starting_z, num scaling)
        VAR robtarget z_0;
        VAR robtarget z_1;
        VAR robtarget z_2;
        VAR robtarget z_3;
        VAR robtarget z_4;
        VAR robtarget z_5;

        z_0:=[[starting_x + 0 * scaling, starting_y + 9 * scaling, starting_z + 20],[0,0,1,0],[0,0,0,0],[9E+09,9E+09,9E+09,9E+09,9E+09,9E+09]];
        z_1:=[[starting_x + 0 * scaling, starting_y + 9 * scaling, starting_z + 0],[0,0,1,0],[0,0,0,0],[9E+09,9E+09,9E+09,9E+09,9E+09,9E+09]];
        z_2:=[[starting_x + 5.5 * scaling, starting_y + 9 * scaling, starting_z + 0],[0,0,1,0],[0,0,0,0],[9E+09,9E+09,9E+09,9E+09,9E+09,9E+09]];
        z_3:=[[starting_x + 0 * scaling, starting_y + 0 * scaling, starting_z + 0],[0,0,1,0],[0,0,0,0],[9E+09,9E+09,9E+09,9E+09,9E+09,9E+09]];
        z_4:=[[starting_x + 6 * scaling, starting_y + 0 * scaling, starting_z + 0],[0,0,1,0],[0,0,0,0],[9E+09,9E+09,9E+09,9E+09,9E+09,9E+09]];
        z_5:=[[starting_x + 6 * scaling, starting_y + 0 * scaling, starting_z + 20],[0,0,1,0],[0,0,0,0],[9E+09,9E+09,9E+09,9E+09,9E+09,9E+09]];

        MoveL z_0,v50,fine,MyNewTool\WObj:=A3;
        MoveL z_1,v50,fine,MyNewTool\WObj:=A3;
        MoveL z_2,v50,fine,MyNewTool\WObj:=A3;
        MoveL z_3,v50,fine,MyNewTool\WObj:=A3;
        MoveL z_4,v50,fine,MyNewTool\WObj:=A3;
        MoveL z_5,v50,fine,MyNewTool\WObj:=A3;

    ENDPROC

    PROC dash(num starting_x, num starting_y, num starting_z, num scaling)
        VAR robtarget dash_0;
        VAR robtarget dash_1;
        VAR robtarget dash_2;
        VAR robtarget dash_3;

        dash_0:=[[starting_x + 0 * scaling, starting_y + 5 * scaling, starting_z + 20],[0,0,1,0],[0,0,0,0],[9E+09,9E+09,9E+09,9E+09,9E+09,9E+09]];
        dash_1:=[[starting_x + 0 * scaling, starting_y + 5 * scaling, starting_z + 0],[0,0,1,0],[0,0,0,0],[9E+09,9E+09,9E+09,9E+09,9E+09,9E+09]];
        dash_2:=[[starting_x + 4.5 * scaling, starting_y + 5 * scaling, starting_z + 0],[0,0,1,0],[0,0,0,0],[9E+09,9E+09,9E+09,9E+09,9E+09,9E+09]];
        dash_3:=[[starting_x + 4.5 * scaling, starting_y + 5 * scaling, starting_z + 20],[0,0,1,0],[0,0,0,0],[9E+09,9E+09,9E+09,9E+09,9E+09,9E+09]];

        MoveL dash_0,v50,fine,MyNewTool\WObj:=A3;
        MoveL dash_1,v50,fine,MyNewTool\WObj:=A3;
        MoveL dash_2,v50,fine,MyNewTool\WObj:=A3;
        MoveL dash_3,v50,fine,MyNewTool\WObj:=A3;

    ENDPROC

    PROC dot(num starting_x, num starting_y, num starting_z, num scaling)
        VAR robtarget dot_0;
        VAR robtarget dot_1;
        VAR robtarget dot_2;
        VAR robtarget dot_3;
        VAR robtarget dot_4;
        VAR robtarget dot_5;
        VAR robtarget dot_6;


        dot_0:=[[starting_x + 0 * scaling, starting_y + 0.75 * scaling, starting_z + 20],[0,0,1,0],[0,0,0,0],[9E+09,9E+09,9E+09,9E+09,9E+09,9E+09]];
        dot_1:=[[starting_x + 0 * scaling, starting_y + 0.75 * scaling, starting_z + 0],[0,0,1,0],[0,0,0,0],[9E+09,9E+09,9E+09,9E+09,9E+09,9E+09]];
        dot_2:=[[starting_x + .75 * scaling, starting_y + 1.5 * scaling, starting_z + 0],[0,0,1,0],[0,0,0,0],[9E+09,9E+09,9E+09,9E+09,9E+09,9E+09]];
        dot_3:=[[starting_x + 1.5 * scaling, starting_y + 0.75 * scaling, starting_z + 0],[0,0,1,0],[0,0,0,0],[9E+09,9E+09,9E+09,9E+09,9E+09,9E+09]];
        dot_4:=[[starting_x + .75 * scaling, starting_y + 0 * scaling, starting_z + 0],[0,0,1,0],[0,0,0,0],[9E+09,9E+09,9E+09,9E+09,9E+09,9E+09]];
        dot_5:=[[starting_x + 0 * scaling, starting_y + 0.75 * scaling, starting_z + 0],[0,0,1,0],[0,0,0,0],[9E+09,9E+09,9E+09,9E+09,9E+09,9E+09]];
        dot_6:=[[starting_x + 0 * scaling, starting_y + 0.75 * scaling, starting_z + 20],[0,0,1,0],[0,0,0,0],[9E+09,9E+09,9E+09,9E+09,9E+09,9E+09]];

        MoveL dot_0,v50,fine,MyNewTool\WObj:=A3;
        MoveL dot_1,v50,fine,MyNewTool\WObj:=A3;
        MoveC dot_2,dot_3,v50,fine,MyNewTool\WObj:=A3;
        MoveC dot_4,dot_5,v50,fine,MyNewTool\WObj:=A3;
        MoveL dot_6,v50,fine,MyNewTool\WObj:=A3;

    ENDPROC

    PROC question(num starting_x, num starting_y, num starting_z, num scaling)
        VAR robtarget question_0;
        VAR robtarget question_1;
        VAR robtarget question_2;
        VAR robtarget question_3;
        VAR robtarget question_4;
        VAR robtarget question_5;
        VAR robtarget question_6;
        VAR robtarget question_7;
        VAR robtarget question_8;
        VAR robtarget question_9;
        VAR robtarget question_10;
        VAR robtarget question_11;
        VAR robtarget question_12;
        VAR robtarget question_13;
        VAR robtarget question_14;

        question_0:=[[starting_x + 0 * scaling, starting_y + 12 * scaling, starting_z + 20],[0,0,1,0],[0,0,0,0],[9E+09,9E+09,9E+09,9E+09,9E+09,9E+09]];
        question_1:=[[starting_x + 0 * scaling, starting_y + 12 * scaling, starting_z + 0],[0,0,1,0],[0,0,0,0],[9E+09,9E+09,9E+09,9E+09,9E+09,9E+09]];
        question_2:=[[starting_x + 3 * scaling, starting_y + 13 * scaling, starting_z + 0],[0,0,1,0],[0,0,0,0],[9E+09,9E+09,9E+09,9E+09,9E+09,9E+09]];
        question_3:=[[starting_x + 6 * scaling, starting_y + 10 * scaling, starting_z + 0],[0,0,1,0],[0,0,0,0],[9E+09,9E+09,9E+09,9E+09,9E+09,9E+09]];
        question_4:=[[starting_x + 5 * scaling, starting_y + 7 * scaling, starting_z + 0],[0,0,1,0],[0,0,0,0],[9E+09,9E+09,9E+09,9E+09,9E+09,9E+09]];
        question_5:=[[starting_x + 2.5 * scaling, starting_y + 6.5 * scaling, starting_z + 0],[0,0,1,0],[0,0,0,0],[9E+09,9E+09,9E+09,9E+09,9E+09,9E+09]];
        question_6:=[[starting_x + 2.5 * scaling, starting_y + 3 * scaling, starting_z + 0],[0,0,1,0],[0,0,0,0],[9E+09,9E+09,9E+09,9E+09,9E+09,9E+09]];
        question_7:=[[starting_x + 2.5 * scaling, starting_y + 3 * scaling, starting_z + 20],[0,0,1,0],[0,0,0,0],[9E+09,9E+09,9E+09,9E+09,9E+09,9E+09]];
        question_8:=[[starting_x + 1.75 * scaling, starting_y + 0.75 * scaling, starting_z + 20],[0,0,1,0],[0,0,0,0],[9E+09,9E+09,9E+09,9E+09,9E+09,9E+09]];
        question_9:=[[starting_x + 1.75 * scaling, starting_y + 0.75 * scaling, starting_z + 0],[0,0,1,0],[0,0,0,0],[9E+09,9E+09,9E+09,9E+09,9E+09,9E+09]];
        question_10:=[[starting_x + 2.5 * scaling, starting_y + 1.5 * scaling, starting_z + 0],[0,0,1,0],[0,0,0,0],[9E+09,9E+09,9E+09,9E+09,9E+09,9E+09]];
        question_11:=[[starting_x + 3.25 * scaling, starting_y + 0.75 * scaling, starting_z + 0],[0,0,1,0],[0,0,0,0],[9E+09,9E+09,9E+09,9E+09,9E+09,9E+09]];
        question_12:=[[starting_x + 2.5 * scaling, starting_y + 0 * scaling, starting_z + 0],[0,0,1,0],[0,0,0,0],[9E+09,9E+09,9E+09,9E+09,9E+09,9E+09]];
        question_13:=[[starting_x + 1.75 * scaling, starting_y + 0.75 * scaling, starting_z + 0],[0,0,1,0],[0,0,0,0],[9E+09,9E+09,9E+09,9E+09,9E+09,9E+09]];
        question_14:=[[starting_x + 1.75 * scaling, starting_y + 0.75 * scaling, starting_z + 20],[0,0,1,0],[0,0,0,0],[9E+09,9E+09,9E+09,9E+09,9E+09,9E+09]];

        MoveL question_0,v50,fine,MyNewTool\WObj:=A3;
        MoveL question_1,v50,fine,MyNewTool\WObj:=A3;
        MoveC question_2,question_3,v50,z5,MyNewTool\WObj:=A3;
        MoveC question_4,question_5,v50,z5,MyNewTool\WObj:=A3;
        MoveL question_6,v50,fine,MyNewTool\WObj:=A3;
        MoveL question_7,v50,fine,MyNewTool\WObj:=A3;
        MoveL question_8,v50,fine,MyNewTool\WObj:=A3;
        MoveL question_9,v50,fine,MyNewTool\WObj:=A3;
        MoveC question_10,question_11,v50,fine,MyNewTool\WObj:=A3;
        MoveC question_12,question_13,v50,fine,MyNewTool\WObj:=A3;
        MoveL question_14,v50,fine,MyNewTool\WObj:=A3;

    ENDPROC


!This procedure writes the initials of the author
	PROC Initials()
	    MoveJ Home_1,v50,fine,MyNewTool\WObj:=A3;
	    MoveL Home_Top_Left_Corner,v50,fine,MyNewTool\WObj:=A3;
	    MoveL Top_of_Start_R,v50,fine,MyNewTool\WObj:=A3;
	    MoveL Start_R,v50,fine,MyNewTool\WObj:=A3;
	    MoveC First_Bottom_curve_R,First_Bottom_curve_R_1,v50,fine,MyNewTool\WObj:=A3;
	    MoveL First_Bottom_curve_R_2,v50,fine,MyNewTool\WObj:=A3;
	    MoveL Line_for_R_and_TCR4,v50,fine,MyNewTool\WObj:=A3;
	    MoveL Top_Line_for_R_and_TCR4,v50,fine,MyNewTool\WObj:=A3;
	    MoveL Top_of_Top_Curve_R,v50,fine,MyNewTool\WObj:=A3;
	    MoveL Top_Curve_R,v50,fine,MyNewTool\WObj:=A3;
	    MoveC Top_Curve_R_1,Top_Curve_R_2,v50,fine,MyNewTool\WObj:=A3;
	    MoveC Top_Curve_R_3,Line_for_R_and_TCR4,v50,fine,MyNewTool\WObj:=A3;
	    MoveC Top_Curve_R_5,Top_Curve_R_6,v50,fine,MyNewTool\WObj:=A3;
	    MoveL Second_Bottom_Curve_R,v50,fine,MyNewTool\WObj:=A3;
	    MoveL Second_Bottom_Curve_R_2,v50,fine,MyNewTool\WObj:=A3;
	    MoveC Second_Bottom_Curve_R_3,Second_Bottom_Curve_R_4,v50,fine,MyNewTool\WObj:=A3;
	    MoveC Second_Bottom_Curve_R_5,Second_Bottom_Curve_R_6,v50,fine,MyNewTool\WObj:=A3;
	    MoveL Second_Bottom_Curve_R_7,v50,fine,MyNewTool\WObj:=A3;
	    MoveC Second_Bottom_Curve_R_8,Finish_R,v50,fine,MyNewTool\WObj:=A3;
	    MoveL Top_of_Finish_R,v50,fine,MyNewTool\WObj:=A3;
	    MoveL Top_of_DOT_R,v50,fine,MyNewTool\WObj:=A3;
	    MoveL DOT_R,v50,fine,MyNewTool\WObj:=A3;
	    MoveC DOT_R_1,DOT_R_2,v50,fine,MyNewTool\WObj:=A3;
	    MoveC DOT_R_3,DOT_R,v50,fine,MyNewTool\WObj:=A3;
	    MoveL Top_of_DOT_R,v50,fine,MyNewTool\WObj:=A3;
	    MoveL Top_of_Start_M,v50,fine,MyNewTool\WObj:=A3;
	    MoveL Start_M,v50,fine,MyNewTool\WObj:=A3;
	    MoveC First_Bottom_curve_M,First_Bottom_curve_M_1,v50,fine,MyNewTool\WObj:=A3;
	    MoveL First_Bottom_curve_M_2,v50,fine,MyNewTool\WObj:=A3;
	    MoveL Line_for_M,v50,fine,MyNewTool\WObj:=A3;
	    MoveL Line_for_M_2,v50,fine,MyNewTool\WObj:=A3;
	    MoveL Line_for_M_3,v50,fine,MyNewTool\WObj:=A3;
	    MoveL Line_for_M_4,v50,fine,MyNewTool\WObj:=A3;
	    MoveL Second_Bottom_Curve_M_1,v50,fine,MyNewTool\WObj:=A3;
	    MoveC Second_Bottom_Curve_M_2,Finish_M,v50,fine,MyNewTool\WObj:=A3;
	    MoveL Top_of_Finish_M,v50,fine,MyNewTool\WObj:=A3;
	    MoveL Top_of_DOT_M,v50,fine,MyNewTool\WObj:=A3;
	    MoveL DOT_M,v50,fine,MyNewTool\WObj:=A3;
	    MoveC DOT_M_1,DOT_M_2,v50,fine,MyNewTool\WObj:=A3;
	    MoveC DOT_M_3,DOT_M,v50,fine,MyNewTool\WObj:=A3;
	    MoveL Top_of_DOT_M,v50,fine,MyNewTool\WObj:=A3;
	    MoveL Home_1,v50,fine,MyNewTool\WObj:=A3;
	ENDPROC

    !The procedures below draw a wolf in the A3 sheet
    PROC Wolf_Outline()
        MoveL Target_10_3,v50,fine,MyNewTool\WObj:=A3;
        MoveL Target_10,v50,fine,MyNewTool\WObj:=A3;
        MoveL Target_20,v50,fine,MyNewTool\WObj:=A3;
        MoveL Target_30,v50,fine,MyNewTool\WObj:=A3;
        MoveL Target_40,v50,fine,MyNewTool\WObj:=A3;
        MoveL Target_50,v50,fine,MyNewTool\WObj:=A3;
        MoveL Target_60,v50,fine,MyNewTool\WObj:=A3;
        MoveL Target_70,v50,fine,MyNewTool\WObj:=A3;
        MoveL Target_80,v50,fine,MyNewTool\WObj:=A3;
        MoveL Target_90,v50,fine,MyNewTool\WObj:=A3;
        MoveL Target_100,v50,fine,MyNewTool\WObj:=A3;
        MoveL Target_110,v50,fine,MyNewTool\WObj:=A3;
        MoveL Target_120,v50,fine,MyNewTool\WObj:=A3;
        MoveL Target_130,v50,fine,MyNewTool\WObj:=A3;
        MoveL Target_140,v50,fine,MyNewTool\WObj:=A3;
        MoveL Target_150,v50,fine,MyNewTool\WObj:=A3;
        MoveL Target_160,v50,fine,MyNewTool\WObj:=A3;
        MoveL Target_170,v50,fine,MyNewTool\WObj:=A3;
        MoveL Target_180,v50,fine,MyNewTool\WObj:=A3;
        MoveL Target_190,v50,fine,MyNewTool\WObj:=A3;
        MoveL Target_200,v50,fine,MyNewTool\WObj:=A3;
        MoveL Target_210,v50,fine,MyNewTool\WObj:=A3;
        MoveL Target_220,v50,fine,MyNewTool\WObj:=A3;
        MoveL Target_230,v50,fine,MyNewTool\WObj:=A3;
        MoveL Target_240,v50,fine,MyNewTool\WObj:=A3;
        MoveL Target_250,v50,fine,MyNewTool\WObj:=A3;
        MoveL Target_260,v50,fine,MyNewTool\WObj:=A3;
        MoveL Target_270,v50,fine,MyNewTool\WObj:=A3;
        MoveL Target_280,v50,fine,MyNewTool\WObj:=A3;
        MoveL Target_290,v50,fine,MyNewTool\WObj:=A3;
        MoveL Target_300,v50,fine,MyNewTool\WObj:=A3;
        MoveL Target_310,v50,fine,MyNewTool\WObj:=A3;
        MoveL Target_320,v50,fine,MyNewTool\WObj:=A3;
        MoveL Target_330,v50,fine,MyNewTool\WObj:=A3;
        MoveL Target_340,v50,fine,MyNewTool\WObj:=A3;
        MoveL Target_350,v50,fine,MyNewTool\WObj:=A3;
        MoveL Target_360,v50,fine,MyNewTool\WObj:=A3;
        MoveL Target_370,v50,fine,MyNewTool\WObj:=A3;
        MoveL Target_380,v50,fine,MyNewTool\WObj:=A3;
        MoveL Target_390,v50,fine,MyNewTool\WObj:=A3;
        MoveL Target_400,v50,fine,MyNewTool\WObj:=A3;
        MoveL Target_410,v50,fine,MyNewTool\WObj:=A3;
        MoveL Target_420,v50,fine,MyNewTool\WObj:=A3;
        MoveL Target_430,v50,fine,MyNewTool\WObj:=A3;
        MoveL Target_440,v50,fine,MyNewTool\WObj:=A3;
        MoveL Target_450,v50,fine,MyNewTool\WObj:=A3;
        MoveL Target_460,v50,fine,MyNewTool\WObj:=A3;
        MoveL Target_470,v50,fine,MyNewTool\WObj:=A3;
        MoveL Target_480,v50,fine,MyNewTool\WObj:=A3;
        MoveL Target_490,v50,fine,MyNewTool\WObj:=A3;
        MoveL Target_500,v50,fine,MyNewTool\WObj:=A3;
        MoveL Target_510,v50,fine,MyNewTool\WObj:=A3;
        MoveL Target_520,v50,fine,MyNewTool\WObj:=A3;
        MoveL Target_530,v50,fine,MyNewTool\WObj:=A3;
        MoveL Target_540,v50,fine,MyNewTool\WObj:=A3;
        MoveL Target_550,v50,fine,MyNewTool\WObj:=A3;
        MoveL Target_560,v50,fine,MyNewTool\WObj:=A3;
        MoveL Target_570,v50,fine,MyNewTool\WObj:=A3;
        MoveL Target_580,v50,fine,MyNewTool\WObj:=A3;
        MoveL Target_590,v50,fine,MyNewTool\WObj:=A3;
        MoveL Target_600,v50,fine,MyNewTool\WObj:=A3;
        MoveL Target_610,v50,fine,MyNewTool\WObj:=A3;
        MoveL Target_620,v50,fine,MyNewTool\WObj:=A3;
        MoveL Target_630,v50,fine,MyNewTool\WObj:=A3;
        MoveL Target_640,v50,fine,MyNewTool\WObj:=A3;
        MoveL Target_650,v50,fine,MyNewTool\WObj:=A3;
        MoveL Target_660,v50,fine,MyNewTool\WObj:=A3;
        MoveL Target_670,v50,fine,MyNewTool\WObj:=A3;
        MoveL Target_680,v50,fine,MyNewTool\WObj:=A3;
        MoveL Target_690,v50,fine,MyNewTool\WObj:=A3;
        MoveL Target_700,v50,fine,MyNewTool\WObj:=A3;
        MoveL Target_710,v50,fine,MyNewTool\WObj:=A3;
        MoveL Target_720,v50,fine,MyNewTool\WObj:=A3;
        MoveL Target_730,v50,fine,MyNewTool\WObj:=A3;
        MoveL Target_740,v50,fine,MyNewTool\WObj:=A3;
        MoveL Target_750,v50,fine,MyNewTool\WObj:=A3;
        MoveL Target_760,v50,fine,MyNewTool\WObj:=A3;
        MoveL Target_770,v50,fine,MyNewTool\WObj:=A3;
        MoveL Target_780,v50,fine,MyNewTool\WObj:=A3;
        MoveL Target_790,v50,fine,MyNewTool\WObj:=A3;
        MoveL Target_800,v50,fine,MyNewTool\WObj:=A3;
        MoveL Target_810,v50,fine,MyNewTool\WObj:=A3;
        MoveL Target_820,v50,fine,MyNewTool\WObj:=A3;
        MoveL Target_830,v50,fine,MyNewTool\WObj:=A3;
        MoveL Target_840,v50,fine,MyNewTool\WObj:=A3;
        MoveL Target_850,v50,fine,MyNewTool\WObj:=A3;
        MoveL Target_860,v50,fine,MyNewTool\WObj:=A3;
        MoveL Target_870,v50,fine,MyNewTool\WObj:=A3;
        MoveL Target_880,v50,fine,MyNewTool\WObj:=A3;
        MoveL Target_890,v50,fine,MyNewTool\WObj:=A3;
        MoveL Target_900,v50,fine,MyNewTool\WObj:=A3;
        MoveL Target_910,v50,fine,MyNewTool\WObj:=A3;
        MoveL Target_920,v50,fine,MyNewTool\WObj:=A3;
        MoveL Target_930,v50,fine,MyNewTool\WObj:=A3;
        MoveL Target_940,v50,fine,MyNewTool\WObj:=A3;
        MoveL Target_950,v50,fine,MyNewTool\WObj:=A3;
        MoveL Target_960,v50,fine,MyNewTool\WObj:=A3;
        MoveL Target_970,v50,fine,MyNewTool\WObj:=A3;
        MoveL Target_980,v50,fine,MyNewTool\WObj:=A3;
        MoveL Target_990,v50,fine,MyNewTool\WObj:=A3;
        MoveL Target_1000,v50,fine,MyNewTool\WObj:=A3;
        MoveL Target_1010,v50,fine,MyNewTool\WObj:=A3;
        MoveL Target_1020,v50,fine,MyNewTool\WObj:=A3;
        MoveL Target_1030,v50,fine,MyNewTool\WObj:=A3;
        MoveL Target_1040,v50,fine,MyNewTool\WObj:=A3;
        MoveL Target_1050,v50,fine,MyNewTool\WObj:=A3;
        MoveL Target_1060,v50,fine,MyNewTool\WObj:=A3;
        MoveL Target_1070,v50,fine,MyNewTool\WObj:=A3;
        MoveL Target_1080,v50,fine,MyNewTool\WObj:=A3;
        MoveL Target_1090,v50,fine,MyNewTool\WObj:=A3;
        MoveL Target_1100,v50,fine,MyNewTool\WObj:=A3;
        MoveL Target_1110,v50,fine,MyNewTool\WObj:=A3;
        MoveL Target_1120,v50,fine,MyNewTool\WObj:=A3;
        MoveL Target_1130,v50,fine,MyNewTool\WObj:=A3;
        MoveL Target_1140,v50,fine,MyNewTool\WObj:=A3;
        MoveL Target_1150,v50,fine,MyNewTool\WObj:=A3;
        MoveL Target_1160,v50,fine,MyNewTool\WObj:=A3;
        MoveL Target_1170,v50,fine,MyNewTool\WObj:=A3;
        MoveL Target_1180,v50,fine,MyNewTool\WObj:=A3;
        MoveL Target_1190,v50,fine,MyNewTool\WObj:=A3;
        MoveL Target_1200,v50,fine,MyNewTool\WObj:=A3;
        MoveL Target_1210,v50,fine,MyNewTool\WObj:=A3;
        MoveL Target_1220,v50,fine,MyNewTool\WObj:=A3;
        MoveL Target_1230,v50,fine,MyNewTool\WObj:=A3;
        MoveL Target_1240,v50,fine,MyNewTool\WObj:=A3;
        MoveL Target_1250,v50,fine,MyNewTool\WObj:=A3;
        MoveL Target_1260,v50,fine,MyNewTool\WObj:=A3;
        MoveL Target_1270,v50,fine,MyNewTool\WObj:=A3;
        MoveL Target_1280,v50,fine,MyNewTool\WObj:=A3;
        MoveL Target_1290,v50,fine,MyNewTool\WObj:=A3;
        MoveL Target_1300,v50,fine,MyNewTool\WObj:=A3;
        MoveL Target_1310,v50,fine,MyNewTool\WObj:=A3;
        MoveL Target_1320,v50,fine,MyNewTool\WObj:=A3;
        MoveL Target_1330,v50,fine,MyNewTool\WObj:=A3;
        MoveL Target_1340,v50,fine,MyNewTool\WObj:=A3;
        MoveL Target_1350,v50,fine,MyNewTool\WObj:=A3;
        MoveL Target_1360,v50,fine,MyNewTool\WObj:=A3;
        MoveL Target_1370,v50,fine,MyNewTool\WObj:=A3;
        MoveL Target_1380,v50,fine,MyNewTool\WObj:=A3;
        MoveL Target_1390,v50,fine,MyNewTool\WObj:=A3;
        MoveL Target_1400,v50,fine,MyNewTool\WObj:=A3;
        MoveL Target_1410,v50,fine,MyNewTool\WObj:=A3;
        MoveL Target_1420,v50,fine,MyNewTool\WObj:=A3;
        MoveL Target_1430,v50,fine,MyNewTool\WObj:=A3;
        MoveL Target_1440,v50,fine,MyNewTool\WObj:=A3;
        MoveL Target_1450,v50,fine,MyNewTool\WObj:=A3;
        MoveL Target_1460,v50,fine,MyNewTool\WObj:=A3;
        MoveL Target_1470,v50,fine,MyNewTool\WObj:=A3;
        MoveL Target_1480,v50,fine,MyNewTool\WObj:=A3;
        MoveL Target_1490,v50,fine,MyNewTool\WObj:=A3;
        MoveL Target_1500,v50,fine,MyNewTool\WObj:=A3;
        MoveL Target_1510,v50,fine,MyNewTool\WObj:=A3;
        MoveL Target_1520,v50,fine,MyNewTool\WObj:=A3;
        MoveL Target_1530,v50,fine,MyNewTool\WObj:=A3;
        MoveL Target_1540,v50,fine,MyNewTool\WObj:=A3;
        MoveL Target_1550,v50,fine,MyNewTool\WObj:=A3;
        MoveL Target_1560,v50,fine,MyNewTool\WObj:=A3;
        MoveL Target_1570,v50,fine,MyNewTool\WObj:=A3;
        MoveL Target_1580,v50,fine,MyNewTool\WObj:=A3;
        MoveL Target_1590,v50,fine,MyNewTool\WObj:=A3;
        MoveL Target_1600,v50,fine,MyNewTool\WObj:=A3;
        MoveL Target_1610,v50,fine,MyNewTool\WObj:=A3;
        MoveL Target_1620,v50,fine,MyNewTool\WObj:=A3;
        MoveL Target_1630,v50,fine,MyNewTool\WObj:=A3;
        MoveL Target_1640,v50,fine,MyNewTool\WObj:=A3;
        MoveL Target_1650,v50,fine,MyNewTool\WObj:=A3;
        MoveL Target_1660,v50,fine,MyNewTool\WObj:=A3;
        MoveL Target_1670,v50,fine,MyNewTool\WObj:=A3;
        MoveL Target_1680,v50,fine,MyNewTool\WObj:=A3;
        MoveL Target_1690,v50,fine,MyNewTool\WObj:=A3;
        MoveL Target_1700,v50,fine,MyNewTool\WObj:=A3;
        MoveL Target_1710,v50,fine,MyNewTool\WObj:=A3;
        MoveL Target_1720,v50,fine,MyNewTool\WObj:=A3;
        MoveL Target_1730,v50,fine,MyNewTool\WObj:=A3;
        MoveL Target_1740,v50,fine,MyNewTool\WObj:=A3;
        MoveL Target_1750,v50,fine,MyNewTool\WObj:=A3;
        MoveL Target_1760,v50,fine,MyNewTool\WObj:=A3;
        MoveL Target_1770,v50,fine,MyNewTool\WObj:=A3;
        MoveL Target_1780,v50,fine,MyNewTool\WObj:=A3;
        MoveL Target_1790,v50,fine,MyNewTool\WObj:=A3;
        MoveL Target_1800,v50,fine,MyNewTool\WObj:=A3;
        MoveL Target_1810,v50,fine,MyNewTool\WObj:=A3;
        MoveL Target_1820,v50,fine,MyNewTool\WObj:=A3;
        MoveL Target_1830,v50,fine,MyNewTool\WObj:=A3;
        MoveL Target_1840,v50,fine,MyNewTool\WObj:=A3;
        MoveL Target_1850,v50,fine,MyNewTool\WObj:=A3;
        MoveL Target_1860,v50,fine,MyNewTool\WObj:=A3;
        MoveL Target_1870,v50,fine,MyNewTool\WObj:=A3;
        MoveL Target_1880,v50,fine,MyNewTool\WObj:=A3;
        MoveL Target_1890,v50,fine,MyNewTool\WObj:=A3;
        MoveL Target_1900,v50,fine,MyNewTool\WObj:=A3;
        MoveL Target_1910,v50,fine,MyNewTool\WObj:=A3;
        MoveL Target_1920,v50,fine,MyNewTool\WObj:=A3;
        MoveL Target_1930,v50,fine,MyNewTool\WObj:=A3;
        MoveL Target_1940,v50,fine,MyNewTool\WObj:=A3;
        MoveL Target_1950,v50,fine,MyNewTool\WObj:=A3;
        MoveL Target_1960,v50,fine,MyNewTool\WObj:=A3;
        MoveL Target_1970,v50,fine,MyNewTool\WObj:=A3;
        MoveL Target_1980,v50,fine,MyNewTool\WObj:=A3;
        MoveL Target_1990,v50,fine,MyNewTool\WObj:=A3;
        MoveL Target_2000,v50,fine,MyNewTool\WObj:=A3;
        MoveL Target_2010,v50,fine,MyNewTool\WObj:=A3;
        MoveL Target_2020,v50,fine,MyNewTool\WObj:=A3;
        MoveL Target_2030,v50,fine,MyNewTool\WObj:=A3;
        MoveL Target_2040,v50,fine,MyNewTool\WObj:=A3;
        MoveL Target_2050,v50,fine,MyNewTool\WObj:=A3;
        MoveL Target_2060,v50,fine,MyNewTool\WObj:=A3;
        MoveL Target_2070,v50,fine,MyNewTool\WObj:=A3;
        MoveL Target_2080,v50,fine,MyNewTool\WObj:=A3;
        MoveL Target_2090,v50,fine,MyNewTool\WObj:=A3;
        MoveL Target_2100,v50,fine,MyNewTool\WObj:=A3;
        MoveL Target_2110,v50,fine,MyNewTool\WObj:=A3;
        MoveL Target_2120,v50,fine,MyNewTool\WObj:=A3;
        MoveL Target_2130,v50,fine,MyNewTool\WObj:=A3;
        MoveL Target_2140,v50,fine,MyNewTool\WObj:=A3;
        MoveL Target_2150,v50,fine,MyNewTool\WObj:=A3;
        MoveL Target_2160,v50,fine,MyNewTool\WObj:=A3;
        MoveL Target_2170,v50,fine,MyNewTool\WObj:=A3;
        MoveL Target_2180,v50,fine,MyNewTool\WObj:=A3;
        MoveL Target_2190,v50,fine,MyNewTool\WObj:=A3;
        MoveL Target_2200,v50,fine,MyNewTool\WObj:=A3;
        MoveL Target_2210,v50,fine,MyNewTool\WObj:=A3;
        MoveL Target_2220,v50,fine,MyNewTool\WObj:=A3;
        MoveL Target_2230,v50,fine,MyNewTool\WObj:=A3;
        MoveL Target_2240,v50,fine,MyNewTool\WObj:=A3;
        MoveL Target_2250,v50,fine,MyNewTool\WObj:=A3;
        MoveL Target_2260,v50,fine,MyNewTool\WObj:=A3;
        MoveL Target_2270,v50,fine,MyNewTool\WObj:=A3;
        MoveL Target_2280,v50,fine,MyNewTool\WObj:=A3;
        MoveL Target_2290,v50,fine,MyNewTool\WObj:=A3;
        MoveL Target_2300,v50,fine,MyNewTool\WObj:=A3;
        MoveL Target_2310,v50,fine,MyNewTool\WObj:=A3;
        MoveL Target_2320,v50,fine,MyNewTool\WObj:=A3;
        MoveL Target_2330,v50,fine,MyNewTool\WObj:=A3;
        MoveL Target_2340,v50,fine,MyNewTool\WObj:=A3;
        MoveL Target_2350,v50,fine,MyNewTool\WObj:=A3;
        MoveL Target_2360,v50,fine,MyNewTool\WObj:=A3;
        MoveL Target_2370,v50,fine,MyNewTool\WObj:=A3;
        MoveL Target_2380,v50,fine,MyNewTool\WObj:=A3;
        MoveL Target_2390,v50,fine,MyNewTool\WObj:=A3;
        MoveL Target_2400,v50,fine,MyNewTool\WObj:=A3;
        MoveL Target_2410,v50,fine,MyNewTool\WObj:=A3;
        MoveL Target_2420,v50,fine,MyNewTool\WObj:=A3;
        MoveL Target_2430,v50,fine,MyNewTool\WObj:=A3;
        MoveL Target_2440,v50,fine,MyNewTool\WObj:=A3;
        MoveL Target_2450,v50,fine,MyNewTool\WObj:=A3;
        MoveL Target_2460,v50,fine,MyNewTool\WObj:=A3;
        MoveL Target_2470,v50,fine,MyNewTool\WObj:=A3;
        MoveL Target_2480,v50,fine,MyNewTool\WObj:=A3;
        MoveL Target_2490,v50,fine,MyNewTool\WObj:=A3;
        MoveL Target_2500,v50,fine,MyNewTool\WObj:=A3;
        MoveL Target_2510,v50,fine,MyNewTool\WObj:=A3;
        MoveL Target_2520,v50,fine,MyNewTool\WObj:=A3;
        MoveL Target_2530,v50,fine,MyNewTool\WObj:=A3;
        MoveL Target_2540,v50,fine,MyNewTool\WObj:=A3;
        MoveL Target_2550,v50,fine,MyNewTool\WObj:=A3;
        MoveL Target_2560,v50,fine,MyNewTool\WObj:=A3;
        MoveL Target_2570,v50,fine,MyNewTool\WObj:=A3;
        MoveL Target_2580,v50,fine,MyNewTool\WObj:=A3;
        MoveL Target_2590,v50,fine,MyNewTool\WObj:=A3;
        MoveL Target_2600,v50,fine,MyNewTool\WObj:=A3;
        MoveL Target_2610,v50,fine,MyNewTool\WObj:=A3;
        MoveL Target_2620,v50,fine,MyNewTool\WObj:=A3;
        MoveL Target_2630,v50,fine,MyNewTool\WObj:=A3;
        MoveL Target_2640,v50,fine,MyNewTool\WObj:=A3;
        MoveL Target_2650,v50,fine,MyNewTool\WObj:=A3;
        MoveL Target_2660,v50,fine,MyNewTool\WObj:=A3;
        MoveL Target_2670,v50,fine,MyNewTool\WObj:=A3;
        MoveL Target_2680,v50,fine,MyNewTool\WObj:=A3;
        MoveL Target_2690,v50,fine,MyNewTool\WObj:=A3;
        MoveL Target_2700,v50,fine,MyNewTool\WObj:=A3;
        MoveL Target_2710,v50,fine,MyNewTool\WObj:=A3;
        MoveL Target_2720,v50,fine,MyNewTool\WObj:=A3;
        MoveL Target_2730,v50,fine,MyNewTool\WObj:=A3;
        MoveL Target_2740,v50,fine,MyNewTool\WObj:=A3;
        MoveL Target_2750,v50,fine,MyNewTool\WObj:=A3;
        MoveL Target_2760,v50,fine,MyNewTool\WObj:=A3;
        MoveL Target_2770,v50,fine,MyNewTool\WObj:=A3;
        MoveL Target_2780,v50,fine,MyNewTool\WObj:=A3;
        MoveL Target_2790,v50,fine,MyNewTool\WObj:=A3;
        MoveL Target_2800,v50,fine,MyNewTool\WObj:=A3;
        MoveL Target_2810,v50,fine,MyNewTool\WObj:=A3;
        MoveL Target_2820,v50,fine,MyNewTool\WObj:=A3;
        MoveL Target_2830,v50,fine,MyNewTool\WObj:=A3;
        MoveL Target_2840,v50,fine,MyNewTool\WObj:=A3;
        MoveL Target_2850,v50,fine,MyNewTool\WObj:=A3;
        MoveL Target_2860,v50,fine,MyNewTool\WObj:=A3;
        MoveL Target_2870,v50,fine,MyNewTool\WObj:=A3;
        MoveL Target_2880,v50,fine,MyNewTool\WObj:=A3;
        MoveL Target_2890,v50,fine,MyNewTool\WObj:=A3;
        MoveL Target_2900,v50,fine,MyNewTool\WObj:=A3;
        MoveL Target_2910,v50,fine,MyNewTool\WObj:=A3;
        MoveL Target_2920,v50,fine,MyNewTool\WObj:=A3;
        MoveL Target_2930,v50,fine,MyNewTool\WObj:=A3;
        MoveL Target_2940,v50,fine,MyNewTool\WObj:=A3;
        MoveL Target_2950,v50,fine,MyNewTool\WObj:=A3;
        MoveL Target_2960,v50,fine,MyNewTool\WObj:=A3;
        MoveL Target_2970,v50,fine,MyNewTool\WObj:=A3;
        MoveL Target_2980,v50,fine,MyNewTool\WObj:=A3;
        MoveL Target_2990,v50,fine,MyNewTool\WObj:=A3;
        MoveL Target_3000,v50,fine,MyNewTool\WObj:=A3;
        MoveL Target_3010,v50,fine,MyNewTool\WObj:=A3;
        MoveL Target_3020,v50,fine,MyNewTool\WObj:=A3;
        MoveL Target_3030,v50,fine,MyNewTool\WObj:=A3;
        MoveL Target_3040,v50,fine,MyNewTool\WObj:=A3;
        MoveL Target_3050,v50,fine,MyNewTool\WObj:=A3;
        MoveL Target_3060,v50,fine,MyNewTool\WObj:=A3;
        MoveL Target_3070,v50,fine,MyNewTool\WObj:=A3;
        MoveL Target_3080,v50,fine,MyNewTool\WObj:=A3;
        MoveL Target_3090,v50,fine,MyNewTool\WObj:=A3;
        MoveL Target_3100,v50,fine,MyNewTool\WObj:=A3;
        MoveL Target_3110,v50,fine,MyNewTool\WObj:=A3;
        MoveL Target_3120,v50,fine,MyNewTool\WObj:=A3;
        MoveL Target_3130,v50,fine,MyNewTool\WObj:=A3;
        MoveL Target_3140,v50,fine,MyNewTool\WObj:=A3;
        MoveL Target_3150,v50,fine,MyNewTool\WObj:=A3;
        MoveL Target_3160,v50,fine,MyNewTool\WObj:=A3;
        MoveL Target_3170,v50,fine,MyNewTool\WObj:=A3;
        MoveL Target_3170_2,v50,fine,MyNewTool\WObj:=A3;
    ENDPROC
    PROC Wolf_Upper()
        MoveL Target_3180_2,v50,fine,MyNewTool\WObj:=A3;
        MoveL Target_3180,v50,fine,MyNewTool\WObj:=A3;
        MoveL Target_3190,v50,fine,MyNewTool\WObj:=A3;
        MoveL Target_3200,v50,fine,MyNewTool\WObj:=A3;
        MoveL Target_3210,v50,fine,MyNewTool\WObj:=A3;
        MoveL Target_3220,v50,fine,MyNewTool\WObj:=A3;
        MoveL Target_3230,v50,fine,MyNewTool\WObj:=A3;
        MoveL Target_3240,v50,fine,MyNewTool\WObj:=A3;
        MoveL Target_3250,v50,fine,MyNewTool\WObj:=A3;
        MoveL Target_3260,v50,fine,MyNewTool\WObj:=A3;
        MoveL Target_3270,v50,fine,MyNewTool\WObj:=A3;
        MoveL Target_3280,v50,fine,MyNewTool\WObj:=A3;
        MoveL Target_3290,v50,fine,MyNewTool\WObj:=A3;
        MoveL Target_3300,v50,fine,MyNewTool\WObj:=A3;
        MoveL Target_3310,v50,fine,MyNewTool\WObj:=A3;
        MoveL Target_3320,v50,fine,MyNewTool\WObj:=A3;
        MoveL Target_3330,v50,fine,MyNewTool\WObj:=A3;
        MoveL Target_3340,v50,fine,MyNewTool\WObj:=A3;
        MoveL Target_3350,v50,fine,MyNewTool\WObj:=A3;
        MoveL Target_3360,v50,fine,MyNewTool\WObj:=A3;
        MoveL Target_3370,v50,fine,MyNewTool\WObj:=A3;
        MoveL Target_3380,v50,fine,MyNewTool\WObj:=A3;
        MoveL Target_3390,v50,fine,MyNewTool\WObj:=A3;
        MoveL Target_3400,v50,fine,MyNewTool\WObj:=A3;
        MoveL Target_3400_2,v50,fine,MyNewTool\WObj:=A3;
    ENDPROC
    PROC Wolf_Upper_2()
        MoveL Target_3410_3,v50,fine,MyNewTool\WObj:=A3;
        MoveL Target_3410,v50,fine,MyNewTool\WObj:=A3;
        MoveL Target_3420,v50,fine,MyNewTool\WObj:=A3;
        MoveL Target_3430,v50,fine,MyNewTool\WObj:=A3;
        MoveL Target_3440,v50,fine,MyNewTool\WObj:=A3;
        MoveL Target_3450,v50,fine,MyNewTool\WObj:=A3;
        MoveL Target_3460,v50,fine,MyNewTool\WObj:=A3;
        MoveL Target_3470,v50,fine,MyNewTool\WObj:=A3;
        MoveL Target_3480,v50,fine,MyNewTool\WObj:=A3;
        MoveL Target_3490,v50,fine,MyNewTool\WObj:=A3;
        MoveL Target_3500,v50,fine,MyNewTool\WObj:=A3;
        MoveL Target_3510,v50,fine,MyNewTool\WObj:=A3;
        MoveL Target_3520,v50,fine,MyNewTool\WObj:=A3;
        MoveL Target_3530,v50,fine,MyNewTool\WObj:=A3;
        MoveL Target_3540,v50,fine,MyNewTool\WObj:=A3;
        MoveL Target_3550,v50,fine,MyNewTool\WObj:=A3;
        MoveL Target_3560,v50,fine,MyNewTool\WObj:=A3;
        MoveL Target_3570,v50,fine,MyNewTool\WObj:=A3;
        MoveL Target_3580,v50,fine,MyNewTool\WObj:=A3;
        MoveL Target_3590,v50,fine,MyNewTool\WObj:=A3;
        MoveL Target_3600,v50,fine,MyNewTool\WObj:=A3;
        MoveL Target_3610,v50,fine,MyNewTool\WObj:=A3;
        MoveL Target_3620,v50,fine,MyNewTool\WObj:=A3;
        MoveL Target_3630,v50,fine,MyNewTool\WObj:=A3;
        MoveL Target_3640,v50,fine,MyNewTool\WObj:=A3;
        MoveL Target_3650,v50,fine,MyNewTool\WObj:=A3;
        MoveL Target_3660,v50,fine,MyNewTool\WObj:=A3;
        MoveL Target_3670,v50,fine,MyNewTool\WObj:=A3;
        MoveL Target_3680,v50,fine,MyNewTool\WObj:=A3;
        MoveL Target_3690,v50,fine,MyNewTool\WObj:=A3;
        MoveL Target_3700,v50,fine,MyNewTool\WObj:=A3;
        MoveL Target_3710,v50,fine,MyNewTool\WObj:=A3;
        MoveL Target_3720,v50,fine,MyNewTool\WObj:=A3;
        MoveL Target_3730,v50,fine,MyNewTool\WObj:=A3;
        MoveL Target_3740,v50,fine,MyNewTool\WObj:=A3;
        MoveL Target_3750,v50,fine,MyNewTool\WObj:=A3;
        MoveL Target_3760,v50,fine,MyNewTool\WObj:=A3;
        MoveL Target_3770,v50,fine,MyNewTool\WObj:=A3;
        MoveL Target_3780,v50,fine,MyNewTool\WObj:=A3;
        MoveL Target_3790,v50,fine,MyNewTool\WObj:=A3;
        MoveL Target_3800,v50,fine,MyNewTool\WObj:=A3;
        MoveL Target_3810,v50,fine,MyNewTool\WObj:=A3;
        MoveL Target_3820,v50,fine,MyNewTool\WObj:=A3;
        MoveL Target_3830,v50,fine,MyNewTool\WObj:=A3;
        MoveL Target_3840,v50,fine,MyNewTool\WObj:=A3;
        MoveL Target_3850,v50,fine,MyNewTool\WObj:=A3;
        MoveL Target_3860,v50,fine,MyNewTool\WObj:=A3;
        MoveL Target_3860_2,v50,fine,MyNewTool\WObj:=A3;
    ENDPROC
    PROC Wolf_Mid()
        MoveL Target_3870_2,v50,fine,MyNewTool\WObj:=A3;
        MoveL Target_3870,v50,fine,MyNewTool\WObj:=A3;
        MoveL Target_3880,v50,fine,MyNewTool\WObj:=A3;
        MoveL Target_3890,v50,fine,MyNewTool\WObj:=A3;
        MoveL Target_3900,v50,fine,MyNewTool\WObj:=A3;
        MoveL Target_3910,v50,fine,MyNewTool\WObj:=A3;
        MoveL Target_3920,v50,fine,MyNewTool\WObj:=A3;
        MoveL Target_3930,v50,fine,MyNewTool\WObj:=A3;
        MoveL Target_3940,v50,fine,MyNewTool\WObj:=A3;
        MoveL Target_3950,v50,fine,MyNewTool\WObj:=A3;
        MoveL Target_3960,v50,fine,MyNewTool\WObj:=A3;
        MoveL Target_3970,v50,fine,MyNewTool\WObj:=A3;
        MoveL Target_3980,v50,fine,MyNewTool\WObj:=A3;
        MoveL Target_3990,v50,fine,MyNewTool\WObj:=A3;
        MoveL Target_4000,v50,fine,MyNewTool\WObj:=A3;
        MoveL Target_4010,v50,fine,MyNewTool\WObj:=A3;
        MoveL Target_4020,v50,fine,MyNewTool\WObj:=A3;
        MoveL Target_4030,v50,fine,MyNewTool\WObj:=A3;
        MoveL Target_4040,v50,fine,MyNewTool\WObj:=A3;
        MoveL Target_4050,v50,fine,MyNewTool\WObj:=A3;
        MoveL Target_4060,v50,fine,MyNewTool\WObj:=A3;
        MoveL Target_4070,v50,fine,MyNewTool\WObj:=A3;
        MoveL Target_4080,v50,fine,MyNewTool\WObj:=A3;
        MoveL Target_4090,v50,fine,MyNewTool\WObj:=A3;
        MoveL Target_4100,v50,fine,MyNewTool\WObj:=A3;
        MoveL Target_4110,v50,fine,MyNewTool\WObj:=A3;
        MoveL Target_4120,v50,fine,MyNewTool\WObj:=A3;
        MoveL Target_4130,v50,fine,MyNewTool\WObj:=A3;
        MoveL Target_4140,v50,fine,MyNewTool\WObj:=A3;
        MoveL Target_4150,v50,fine,MyNewTool\WObj:=A3;
        MoveL Target_4160,v50,fine,MyNewTool\WObj:=A3;
        MoveL Target_4170,v50,fine,MyNewTool\WObj:=A3;
        MoveL Target_4180,v50,fine,MyNewTool\WObj:=A3;
        MoveL Target_4190,v50,fine,MyNewTool\WObj:=A3;
        MoveL Target_4200,v50,fine,MyNewTool\WObj:=A3;
        MoveL Target_4210,v50,fine,MyNewTool\WObj:=A3;
        MoveL Target_4220,v50,fine,MyNewTool\WObj:=A3;
        MoveL Target_4230,v50,fine,MyNewTool\WObj:=A3;
        MoveL Target_4240,v50,fine,MyNewTool\WObj:=A3;
        MoveL Target_4250,v50,fine,MyNewTool\WObj:=A3;
        MoveL Target_4260,v50,fine,MyNewTool\WObj:=A3;
        MoveL Target_4270,v50,fine,MyNewTool\WObj:=A3;
        MoveL Target_4280,v50,fine,MyNewTool\WObj:=A3;
        MoveL Target_4290,v50,fine,MyNewTool\WObj:=A3;
        MoveL Target_4300,v50,fine,MyNewTool\WObj:=A3;
        MoveL Target_4310,v50,fine,MyNewTool\WObj:=A3;
        MoveL Target_4320,v50,fine,MyNewTool\WObj:=A3;
        MoveL Target_4330,v50,fine,MyNewTool\WObj:=A3;
        MoveL Target_4340,v50,fine,MyNewTool\WObj:=A3;
        MoveL Target_4350,v50,fine,MyNewTool\WObj:=A3;
        MoveL Target_4360,v50,fine,MyNewTool\WObj:=A3;
        MoveL Target_4370,v50,fine,MyNewTool\WObj:=A3;
        MoveL Target_4380,v50,fine,MyNewTool\WObj:=A3;
        MoveL Target_4390,v50,fine,MyNewTool\WObj:=A3;
        MoveL Target_4400,v50,fine,MyNewTool\WObj:=A3;
        MoveL Target_4410,v50,fine,MyNewTool\WObj:=A3;
        MoveL Target_4420,v50,fine,MyNewTool\WObj:=A3;
        MoveL Target_4430,v50,fine,MyNewTool\WObj:=A3;
        MoveL Target_4440,v50,fine,MyNewTool\WObj:=A3;
        MoveL Target_4450,v50,fine,MyNewTool\WObj:=A3;
        MoveL Target_4460,v50,fine,MyNewTool\WObj:=A3;
        MoveL Target_4470,v50,fine,MyNewTool\WObj:=A3;
        MoveL Target_4480,v50,fine,MyNewTool\WObj:=A3;
        MoveL Target_4490,v50,fine,MyNewTool\WObj:=A3;
        MoveL Target_4500,v50,fine,MyNewTool\WObj:=A3;
        MoveL Target_4510,v50,fine,MyNewTool\WObj:=A3;
        MoveL Target_4520,v50,fine,MyNewTool\WObj:=A3;
        MoveL Target_4530,v50,fine,MyNewTool\WObj:=A3;
        MoveL Target_4540,v50,fine,MyNewTool\WObj:=A3;
        MoveL Target_4550,v50,fine,MyNewTool\WObj:=A3;
        MoveL Target_4560,v50,fine,MyNewTool\WObj:=A3;
        MoveL Target_4570,v50,fine,MyNewTool\WObj:=A3;
        MoveL Target_4580,v50,fine,MyNewTool\WObj:=A3;
        MoveL Target_4590,v50,fine,MyNewTool\WObj:=A3;
        MoveL Target_4600,v50,fine,MyNewTool\WObj:=A3;
        MoveL Target_4610,v50,fine,MyNewTool\WObj:=A3;
        MoveL Target_4620,v50,fine,MyNewTool\WObj:=A3;
        MoveL Target_4630,v50,fine,MyNewTool\WObj:=A3;
        MoveL Target_4640,v50,fine,MyNewTool\WObj:=A3;
        MoveL Target_4650,v50,fine,MyNewTool\WObj:=A3;
        MoveL Target_4660,v50,fine,MyNewTool\WObj:=A3;
        MoveL Target_4670,v50,fine,MyNewTool\WObj:=A3;
        MoveL Target_4680,v50,fine,MyNewTool\WObj:=A3;
        MoveL Target_4690,v50,fine,MyNewTool\WObj:=A3;
        MoveL Target_4700,v50,fine,MyNewTool\WObj:=A3;
        MoveL Target_4710,v50,fine,MyNewTool\WObj:=A3;
        MoveL Target_4720,v50,fine,MyNewTool\WObj:=A3;
        MoveL Target_4730,v50,fine,MyNewTool\WObj:=A3;
        MoveL Target_4740,v50,fine,MyNewTool\WObj:=A3;
        MoveL Target_4750,v50,fine,MyNewTool\WObj:=A3;
        MoveL Target_4760,v50,fine,MyNewTool\WObj:=A3;
        MoveL Target_4770,v50,fine,MyNewTool\WObj:=A3;
        MoveL Target_4780,v50,fine,MyNewTool\WObj:=A3;
        MoveL Target_4790,v50,fine,MyNewTool\WObj:=A3;
        MoveL Target_4800,v50,fine,MyNewTool\WObj:=A3;
        MoveL Target_4810,v50,fine,MyNewTool\WObj:=A3;
        MoveL Target_4820,v50,fine,MyNewTool\WObj:=A3;
        MoveL Target_4830,v50,fine,MyNewTool\WObj:=A3;
        MoveL Target_4840,v50,fine,MyNewTool\WObj:=A3;
        MoveL Target_4850,v50,fine,MyNewTool\WObj:=A3;
        MoveL Target_4860,v50,fine,MyNewTool\WObj:=A3;
        MoveL Target_4870,v50,fine,MyNewTool\WObj:=A3;
        MoveL Target_4880,v50,fine,MyNewTool\WObj:=A3;
        MoveL Target_4890,v50,fine,MyNewTool\WObj:=A3;
        MoveL Target_4900,v50,fine,MyNewTool\WObj:=A3;
        MoveL Target_4910,v50,fine,MyNewTool\WObj:=A3;
        MoveL Target_4920,v50,fine,MyNewTool\WObj:=A3;
        MoveL Target_4930,v50,fine,MyNewTool\WObj:=A3;
        MoveL Target_4940,v50,fine,MyNewTool\WObj:=A3;
        MoveL Target_4950,v50,fine,MyNewTool\WObj:=A3;
        MoveL Target_4960,v50,fine,MyNewTool\WObj:=A3;
        MoveL Target_4970,v50,fine,MyNewTool\WObj:=A3;
        MoveL Target_4980,v50,fine,MyNewTool\WObj:=A3;
        MoveL Target_4990,v50,fine,MyNewTool\WObj:=A3;
        MoveL Target_4990_2,v50,fine,MyNewTool\WObj:=A3;
    ENDPROC
    PROC Wolf_Lower()
        MoveL Target_5000_2,v50,fine,MyNewTool\WObj:=A3;
        MoveL Target_5000,v50,fine,MyNewTool\WObj:=A3;
        MoveL Target_5010,v50,fine,MyNewTool\WObj:=A3;
        MoveL Target_5020,v50,fine,MyNewTool\WObj:=A3;
        MoveL Target_5030,v50,fine,MyNewTool\WObj:=A3;
        MoveL Target_5040,v50,fine,MyNewTool\WObj:=A3;
        MoveL Target_5050,v50,fine,MyNewTool\WObj:=A3;
        MoveL Target_5060,v50,fine,MyNewTool\WObj:=A3;
        MoveL Target_5070,v50,fine,MyNewTool\WObj:=A3;
        MoveL Target_5080,v50,fine,MyNewTool\WObj:=A3;
        MoveL Target_5090,v50,fine,MyNewTool\WObj:=A3;
        MoveL Target_5100,v50,fine,MyNewTool\WObj:=A3;
        MoveL Target_5110,v50,fine,MyNewTool\WObj:=A3;
        MoveL Target_5120,v50,fine,MyNewTool\WObj:=A3;
        MoveL Target_5130,v50,fine,MyNewTool\WObj:=A3;
        MoveL Target_5140,v50,fine,MyNewTool\WObj:=A3;
        MoveL Target_5150,v50,fine,MyNewTool\WObj:=A3;
        MoveL Target_5160,v50,fine,MyNewTool\WObj:=A3;
        MoveL Target_5170,v50,fine,MyNewTool\WObj:=A3;
        MoveL Target_5180,v50,fine,MyNewTool\WObj:=A3;
        MoveL Target_5190,v50,fine,MyNewTool\WObj:=A3;
        MoveL Target_5200,v50,fine,MyNewTool\WObj:=A3;
        MoveL Target_5210,v50,fine,MyNewTool\WObj:=A3;
        MoveL Target_5220,v50,fine,MyNewTool\WObj:=A3;
        MoveL Target_5230,v50,fine,MyNewTool\WObj:=A3;
        MoveL Target_5240,v50,fine,MyNewTool\WObj:=A3;
        MoveL Target_5250,v50,fine,MyNewTool\WObj:=A3;
        MoveL Target_5260,v50,fine,MyNewTool\WObj:=A3;
        MoveL Target_5270,v50,fine,MyNewTool\WObj:=A3;
        MoveL Target_5280,v50,fine,MyNewTool\WObj:=A3;
        MoveL Target_5290,v50,fine,MyNewTool\WObj:=A3;
        MoveL Target_5300,v50,fine,MyNewTool\WObj:=A3;
        MoveL Target_5310,v50,fine,MyNewTool\WObj:=A3;
        MoveL Target_5320,v50,fine,MyNewTool\WObj:=A3;
        MoveL Target_5330,v50,fine,MyNewTool\WObj:=A3;
        MoveL Target_5340,v50,fine,MyNewTool\WObj:=A3;
        MoveL Target_5350,v50,fine,MyNewTool\WObj:=A3;
        MoveL Target_5360,v50,fine,MyNewTool\WObj:=A3;
        MoveL Target_5370,v50,fine,MyNewTool\WObj:=A3;
        MoveL Target_5380,v50,fine,MyNewTool\WObj:=A3;
        MoveL Target_5390,v50,fine,MyNewTool\WObj:=A3;
        MoveL Target_5400,v50,fine,MyNewTool\WObj:=A3;
        MoveL Target_5410,v50,fine,MyNewTool\WObj:=A3;
        MoveL Target_5420,v50,fine,MyNewTool\WObj:=A3;
        MoveL Target_5430,v50,fine,MyNewTool\WObj:=A3;
        MoveL Target_5440,v50,fine,MyNewTool\WObj:=A3;
        MoveL Target_5450,v50,fine,MyNewTool\WObj:=A3;
        MoveL Target_5460,v50,fine,MyNewTool\WObj:=A3;
        MoveL Target_5470,v50,fine,MyNewTool\WObj:=A3;
        MoveL Target_5480,v50,fine,MyNewTool\WObj:=A3;
        MoveL Target_5490,v50,fine,MyNewTool\WObj:=A3;
        MoveL Target_5500,v50,fine,MyNewTool\WObj:=A3;
        MoveL Target_5510,v50,fine,MyNewTool\WObj:=A3;
        MoveL Target_5520,v50,fine,MyNewTool\WObj:=A3;
        MoveL Target_5530,v50,fine,MyNewTool\WObj:=A3;
        MoveL Target_5540,v50,fine,MyNewTool\WObj:=A3;
        MoveL Target_5550,v50,fine,MyNewTool\WObj:=A3;
        MoveL Target_5560,v50,fine,MyNewTool\WObj:=A3;
        MoveL Target_5570,v50,fine,MyNewTool\WObj:=A3;
        MoveL Target_5580,v50,fine,MyNewTool\WObj:=A3;
        MoveL Target_5590,v50,fine,MyNewTool\WObj:=A3;
        MoveL Target_5600,v50,fine,MyNewTool\WObj:=A3;
        MoveL Target_5610,v50,fine,MyNewTool\WObj:=A3;
        MoveL Target_5610_2,v50,fine,MyNewTool\WObj:=A3;
    ENDPROC
    PROC Wolf_Paw()
        MoveL Target_5620_2,v50,fine,MyNewTool\WObj:=A3;
        MoveL Target_5620,v50,fine,MyNewTool\WObj:=A3;
        MoveL Target_5630,v50,fine,MyNewTool\WObj:=A3;
        MoveL Target_5640,v50,fine,MyNewTool\WObj:=A3;
        MoveL Target_5650,v50,fine,MyNewTool\WObj:=A3;
        MoveL Target_5660,v50,fine,MyNewTool\WObj:=A3;
        MoveL Target_5670,v50,fine,MyNewTool\WObj:=A3;
        MoveL Target_5680,v50,fine,MyNewTool\WObj:=A3;
        MoveL Target_5690,v50,fine,MyNewTool\WObj:=A3;
        MoveL Target_5700,v50,fine,MyNewTool\WObj:=A3;
        MoveL Target_5710,v50,fine,MyNewTool\WObj:=A3;
        MoveL Target_5720,v50,fine,MyNewTool\WObj:=A3;
        MoveL Target_5730,v50,fine,MyNewTool\WObj:=A3;
        MoveL Target_5740,v50,fine,MyNewTool\WObj:=A3;
        MoveL Target_5750,v50,fine,MyNewTool\WObj:=A3;
        MoveL Target_5760,v50,fine,MyNewTool\WObj:=A3;
        MoveL Target_5770,v50,fine,MyNewTool\WObj:=A3;
        MoveL Target_5780,v50,fine,MyNewTool\WObj:=A3;
        MoveL Target_5790,v50,fine,MyNewTool\WObj:=A3;
        MoveL Target_5800,v50,fine,MyNewTool\WObj:=A3;
        MoveL Target_5810,v50,fine,MyNewTool\WObj:=A3;
        MoveL Target_5820,v50,fine,MyNewTool\WObj:=A3;
        MoveL Target_5830,v50,fine,MyNewTool\WObj:=A3;
        MoveL Target_5840,v50,fine,MyNewTool\WObj:=A3;
        MoveL Target_5850,v50,fine,MyNewTool\WObj:=A3;
        MoveL Target_5860,v50,fine,MyNewTool\WObj:=A3;
        MoveL Target_5870,v50,fine,MyNewTool\WObj:=A3;
        MoveL Target_5880,v50,fine,MyNewTool\WObj:=A3;
        MoveL Target_5890,v50,fine,MyNewTool\WObj:=A3;
        MoveL Target_5900,v50,fine,MyNewTool\WObj:=A3;
        MoveL Target_5910,v50,fine,MyNewTool\WObj:=A3;
        MoveL Target_5920,v50,fine,MyNewTool\WObj:=A3;
        MoveL Target_5930,v50,fine,MyNewTool\WObj:=A3;
        MoveL Target_5940,v50,fine,MyNewTool\WObj:=A3;
        MoveL Target_5950,v50,fine,MyNewTool\WObj:=A3;
        MoveL Target_5960,v50,fine,MyNewTool\WObj:=A3;
        MoveL Target_5970,v50,fine,MyNewTool\WObj:=A3;
        MoveL Target_5980,v50,fine,MyNewTool\WObj:=A3;
        MoveL Target_5990,v50,fine,MyNewTool\WObj:=A3;
        MoveL Target_6000,v50,fine,MyNewTool\WObj:=A3;
        MoveL Target_6010,v50,fine,MyNewTool\WObj:=A3;
        MoveL Target_6020,v50,fine,MyNewTool\WObj:=A3;
        MoveL Target_6030,v50,fine,MyNewTool\WObj:=A3;
        MoveL Target_6040,v50,fine,MyNewTool\WObj:=A3;
        MoveL Target_6050,v50,fine,MyNewTool\WObj:=A3;
        MoveL Target_6060,v50,fine,MyNewTool\WObj:=A3;
        MoveL Target_6070,v50,fine,MyNewTool\WObj:=A3;
        MoveL Target_6080,v50,fine,MyNewTool\WObj:=A3;
        MoveL Target_6090,v50,fine,MyNewTool\WObj:=A3;
        MoveL Target_6100,v50,fine,MyNewTool\WObj:=A3;
        MoveL Target_6110,v50,fine,MyNewTool\WObj:=A3;
        MoveL Target_6120,v50,fine,MyNewTool\WObj:=A3;
        MoveL Target_6130,v50,fine,MyNewTool\WObj:=A3;
        MoveL Target_6140,v50,fine,MyNewTool\WObj:=A3;
        MoveL Target_6150,v50,fine,MyNewTool\WObj:=A3;
        MoveL Target_6160,v50,fine,MyNewTool\WObj:=A3;
        MoveL Target_6170,v50,fine,MyNewTool\WObj:=A3;
        MoveL Target_6180,v50,fine,MyNewTool\WObj:=A3;
        MoveL Target_6190,v50,fine,MyNewTool\WObj:=A3;
        MoveL Target_6200,v50,fine,MyNewTool\WObj:=A3;
        MoveL Target_6210,v50,fine,MyNewTool\WObj:=A3;
        MoveL Target_6220,v50,fine,MyNewTool\WObj:=A3;
        MoveL Target_6230,v50,fine,MyNewTool\WObj:=A3;
        MoveL Target_6240,v50,fine,MyNewTool\WObj:=A3;
        MoveL Target_6250,v50,fine,MyNewTool\WObj:=A3;
        MoveL Target_6260,v50,fine,MyNewTool\WObj:=A3;
        MoveL Target_6270,v50,fine,MyNewTool\WObj:=A3;
        MoveL Target_6280,v50,fine,MyNewTool\WObj:=A3;
        MoveL Target_6290,v50,fine,MyNewTool\WObj:=A3;
        MoveL Target_6300,v50,fine,MyNewTool\WObj:=A3;
        MoveL Target_6310,v50,fine,MyNewTool\WObj:=A3;
        MoveL Target_6320,v50,fine,MyNewTool\WObj:=A3;
        MoveL Target_6330,v50,fine,MyNewTool\WObj:=A3;
        MoveL Target_6340,v50,fine,MyNewTool\WObj:=A3;
        MoveL Target_6350,v50,fine,MyNewTool\WObj:=A3;
        MoveL Target_6360,v50,fine,MyNewTool\WObj:=A3;
        MoveL Target_6360_2,v50,fine,MyNewTool\WObj:=A3;
    ENDPROC
    PROC Wolf_Paw_2()
        MoveL Target_6370_2,v50,fine,MyNewTool\WObj:=A3;
        MoveL Target_6370,v50,fine,MyNewTool\WObj:=A3;
        MoveL Target_6380,v50,fine,MyNewTool\WObj:=A3;
        MoveL Target_6390,v50,fine,MyNewTool\WObj:=A3;
        MoveL Target_6400,v50,fine,MyNewTool\WObj:=A3;
        MoveL Target_6410,v50,fine,MyNewTool\WObj:=A3;
        MoveL Target_6420,v50,fine,MyNewTool\WObj:=A3;
        MoveL Target_6430,v50,fine,MyNewTool\WObj:=A3;
        MoveL Target_6430_2,v50,fine,MyNewTool\WObj:=A3;
    ENDPROC
    PROC Wolf_Paw_3()
        MoveL Target_6440_2,v50,fine,MyNewTool\WObj:=A3;
        MoveL Target_6440,v50,fine,MyNewTool\WObj:=A3;
        MoveL Target_6450,v50,fine,MyNewTool\WObj:=A3;
        MoveL Target_6460,v50,fine,MyNewTool\WObj:=A3;
        MoveL Target_6470,v50,fine,MyNewTool\WObj:=A3;
        MoveL Target_6480,v50,fine,MyNewTool\WObj:=A3;
        MoveL Target_6490,v50,fine,MyNewTool\WObj:=A3;
        MoveL Target_6500,v50,fine,MyNewTool\WObj:=A3;
        MoveL Target_6510,v50,fine,MyNewTool\WObj:=A3;
        MoveL Target_6520,v50,fine,MyNewTool\WObj:=A3;
        MoveL Target_6530,v50,fine,MyNewTool\WObj:=A3;
        MoveL Target_6530_2,v50,fine,MyNewTool\WObj:=A3;
    ENDPROC
    PROC Wolf_Lower_2()
        MoveL Target_6540_2,v50,fine,MyNewTool\WObj:=A3;
        MoveL Target_6540,v50,fine,MyNewTool\WObj:=A3;
        MoveL Target_6550,v50,fine,MyNewTool\WObj:=A3;
        MoveL Target_6560,v50,fine,MyNewTool\WObj:=A3;
        MoveL Target_6570,v50,fine,MyNewTool\WObj:=A3;
        MoveL Target_6580,v50,fine,MyNewTool\WObj:=A3;
        MoveL Target_6590,v50,fine,MyNewTool\WObj:=A3;
        MoveL Target_6600,v50,fine,MyNewTool\WObj:=A3;
        MoveL Target_6610,v50,fine,MyNewTool\WObj:=A3;
        MoveL Target_6620,v50,fine,MyNewTool\WObj:=A3;
        MoveL Target_6630,v50,fine,MyNewTool\WObj:=A3;
        MoveL Target_6640,v50,fine,MyNewTool\WObj:=A3;
        MoveL Target_6650,v50,fine,MyNewTool\WObj:=A3;
        MoveL Target_6660,v50,fine,MyNewTool\WObj:=A3;
        MoveL Target_6670,v50,fine,MyNewTool\WObj:=A3;
        MoveL Target_6680,v50,fine,MyNewTool\WObj:=A3;
        MoveL Target_6690,v50,fine,MyNewTool\WObj:=A3;
        MoveL Target_6700,v50,fine,MyNewTool\WObj:=A3;
        MoveL Target_6710,v50,fine,MyNewTool\WObj:=A3;
        MoveL Target_6720,v50,fine,MyNewTool\WObj:=A3;
        MoveL Target_6730,v50,fine,MyNewTool\WObj:=A3;
        MoveL Target_6740,v50,fine,MyNewTool\WObj:=A3;
        MoveL Target_6750,v50,fine,MyNewTool\WObj:=A3;
        MoveL Target_6760,v50,fine,MyNewTool\WObj:=A3;
        MoveL Target_6770,v50,fine,MyNewTool\WObj:=A3;
        MoveL Target_6780,v50,fine,MyNewTool\WObj:=A3;
        MoveL Target_6790,v50,fine,MyNewTool\WObj:=A3;
        MoveL Target_6800,v50,fine,MyNewTool\WObj:=A3;
        MoveL Target_6810,v50,fine,MyNewTool\WObj:=A3;
        MoveL Target_6820,v50,fine,MyNewTool\WObj:=A3;
        MoveL Target_6830,v50,fine,MyNewTool\WObj:=A3;
        MoveL Target_6840,v50,fine,MyNewTool\WObj:=A3;
        MoveL Target_6850,v50,fine,MyNewTool\WObj:=A3;
        MoveL Target_6860,v50,fine,MyNewTool\WObj:=A3;
        MoveL Target_6870,v50,fine,MyNewTool\WObj:=A3;
        MoveL Target_6880,v50,fine,MyNewTool\WObj:=A3;
        MoveL Target_6890,v50,fine,MyNewTool\WObj:=A3;
        MoveL Target_6900,v50,fine,MyNewTool\WObj:=A3;
        MoveL Target_6910,v50,fine,MyNewTool\WObj:=A3;
        MoveL Target_6920,v50,fine,MyNewTool\WObj:=A3;
        MoveL Target_6930,v50,fine,MyNewTool\WObj:=A3;
        MoveL Target_6940,v50,fine,MyNewTool\WObj:=A3;
        MoveL Target_6950,v50,fine,MyNewTool\WObj:=A3;
        MoveL Target_6960,v50,fine,MyNewTool\WObj:=A3;
        MoveL Target_6970,v50,fine,MyNewTool\WObj:=A3;
        MoveL Target_6980,v50,fine,MyNewTool\WObj:=A3;
        MoveL Target_6990,v50,fine,MyNewTool\WObj:=A3;
        MoveL Target_7000,v50,fine,MyNewTool\WObj:=A3;
        MoveL Target_7010,v50,fine,MyNewTool\WObj:=A3;
        MoveL Target_7020,v50,fine,MyNewTool\WObj:=A3;
        MoveL Target_7030,v50,fine,MyNewTool\WObj:=A3;
        MoveL Target_7040,v50,fine,MyNewTool\WObj:=A3;
        MoveL Target_7050,v50,fine,MyNewTool\WObj:=A3;
        MoveL Target_7060,v50,fine,MyNewTool\WObj:=A3;
        MoveL Target_7070,v50,fine,MyNewTool\WObj:=A3;
        MoveL Target_7080,v50,fine,MyNewTool\WObj:=A3;
        MoveL Target_7090,v50,fine,MyNewTool\WObj:=A3;
        MoveL Target_7100,v50,fine,MyNewTool\WObj:=A3;
        MoveL Target_7110,v50,fine,MyNewTool\WObj:=A3;
        MoveL Target_7120,v50,fine,MyNewTool\WObj:=A3;
        MoveL Target_7130,v50,fine,MyNewTool\WObj:=A3;
        MoveL Target_7140,v50,fine,MyNewTool\WObj:=A3;
        MoveL Target_7150,v50,fine,MyNewTool\WObj:=A3;
        MoveL Target_7160,v50,fine,MyNewTool\WObj:=A3;
        MoveL Target_7170,v50,fine,MyNewTool\WObj:=A3;
        MoveL Target_7180,v50,fine,MyNewTool\WObj:=A3;
        MoveL Target_7190,v50,fine,MyNewTool\WObj:=A3;
        MoveL Target_7200,v50,fine,MyNewTool\WObj:=A3;
        MoveL Target_7210,v50,fine,MyNewTool\WObj:=A3;
        MoveL Target_7220,v50,fine,MyNewTool\WObj:=A3;
        MoveL Target_7230,v50,fine,MyNewTool\WObj:=A3;
        MoveL Target_7240,v50,fine,MyNewTool\WObj:=A3;
        MoveL Target_7250,v50,fine,MyNewTool\WObj:=A3;
        MoveL Target_7260,v50,fine,MyNewTool\WObj:=A3;
        MoveL Target_7270,v50,fine,MyNewTool\WObj:=A3;
        MoveL Target_7280,v50,fine,MyNewTool\WObj:=A3;
        MoveL Target_7290,v50,fine,MyNewTool\WObj:=A3;
        MoveL Target_7300,v50,fine,MyNewTool\WObj:=A3;
        MoveL Target_7310,v50,fine,MyNewTool\WObj:=A3;
        MoveL Target_7320,v50,fine,MyNewTool\WObj:=A3;
        MoveL Target_7330,v50,fine,MyNewTool\WObj:=A3;
        MoveL Target_7330_2,v50,fine,MyNewTool\WObj:=A3;
    ENDPROC
    PROC Wolf_Outline_2()
        MoveL Target_7340_2,v50,fine,MyNewTool\WObj:=A3;
        MoveL Target_7340,v50,fine,MyNewTool\WObj:=A3;
        MoveL Target_7350,v50,fine,MyNewTool\WObj:=A3;
        MoveL Target_7360,v50,fine,MyNewTool\WObj:=A3;
        MoveL Target_7370,v50,fine,MyNewTool\WObj:=A3;
        MoveL Target_7380,v50,fine,MyNewTool\WObj:=A3;
        MoveL Target_7390,v50,fine,MyNewTool\WObj:=A3;
        MoveL Target_7400,v50,fine,MyNewTool\WObj:=A3;
        MoveL Target_7410,v50,fine,MyNewTool\WObj:=A3;
        MoveL Target_7420,v50,fine,MyNewTool\WObj:=A3;
        MoveL Target_7430,v50,fine,MyNewTool\WObj:=A3;
        MoveL Target_7440,v50,fine,MyNewTool\WObj:=A3;
        MoveL Target_7450,v50,fine,MyNewTool\WObj:=A3;
        MoveL Target_7460,v50,fine,MyNewTool\WObj:=A3;
        MoveL Target_7470,v50,fine,MyNewTool\WObj:=A3;
        MoveL Target_7480,v50,fine,MyNewTool\WObj:=A3;
        MoveL Target_7490,v50,fine,MyNewTool\WObj:=A3;
        MoveL Target_7500,v50,fine,MyNewTool\WObj:=A3;
        MoveL Target_7510,v50,fine,MyNewTool\WObj:=A3;
        MoveL Target_7520,v50,fine,MyNewTool\WObj:=A3;
        MoveL Target_7530,v50,fine,MyNewTool\WObj:=A3;
        MoveL Target_7540,v50,fine,MyNewTool\WObj:=A3;
        MoveL Target_7550,v50,fine,MyNewTool\WObj:=A3;
        MoveL Target_7560,v50,fine,MyNewTool\WObj:=A3;
        MoveL Target_7570,v50,fine,MyNewTool\WObj:=A3;
        MoveL Target_7580,v50,fine,MyNewTool\WObj:=A3;
        MoveL Target_7590,v50,fine,MyNewTool\WObj:=A3;
        MoveL Target_7600,v50,fine,MyNewTool\WObj:=A3;
        MoveL Target_7610,v50,fine,MyNewTool\WObj:=A3;
        MoveL Target_7620,v50,fine,MyNewTool\WObj:=A3;
        MoveL Target_7630,v50,fine,MyNewTool\WObj:=A3;
        MoveL Target_7640,v50,fine,MyNewTool\WObj:=A3;
        MoveL Target_7650,v50,fine,MyNewTool\WObj:=A3;
        MoveL Target_7660,v50,fine,MyNewTool\WObj:=A3;
        MoveL Target_7670,v50,fine,MyNewTool\WObj:=A3;
        MoveL Target_7680,v50,fine,MyNewTool\WObj:=A3;
        MoveL Target_7690,v50,fine,MyNewTool\WObj:=A3;
        MoveL Target_7700,v50,fine,MyNewTool\WObj:=A3;
        MoveL Target_7710,v50,fine,MyNewTool\WObj:=A3;
        MoveL Target_7720,v50,fine,MyNewTool\WObj:=A3;
        MoveL Target_7730,v50,fine,MyNewTool\WObj:=A3;
        MoveL Target_7740,v50,fine,MyNewTool\WObj:=A3;
        MoveL Target_7750,v50,fine,MyNewTool\WObj:=A3;
        MoveL Target_7760,v50,fine,MyNewTool\WObj:=A3;
        MoveL Target_7770,v50,fine,MyNewTool\WObj:=A3;
        MoveL Target_7780,v50,fine,MyNewTool\WObj:=A3;
        MoveL Target_7790,v50,fine,MyNewTool\WObj:=A3;
        MoveL Target_7800,v50,fine,MyNewTool\WObj:=A3;
        MoveL Target_7810,v50,fine,MyNewTool\WObj:=A3;
        MoveL Target_7820,v50,fine,MyNewTool\WObj:=A3;
        MoveL Target_7830,v50,fine,MyNewTool\WObj:=A3;
        MoveL Target_7840,v50,fine,MyNewTool\WObj:=A3;
        MoveL Target_7850,v50,fine,MyNewTool\WObj:=A3;
        MoveL Target_7860,v50,fine,MyNewTool\WObj:=A3;
        MoveL Target_7870,v50,fine,MyNewTool\WObj:=A3;
        MoveL Target_7880,v50,fine,MyNewTool\WObj:=A3;
        MoveL Target_7890,v50,fine,MyNewTool\WObj:=A3;
        MoveL Target_7900,v50,fine,MyNewTool\WObj:=A3;
        MoveL Target_7910,v50,fine,MyNewTool\WObj:=A3;
        MoveL Target_7920,v50,fine,MyNewTool\WObj:=A3;
        MoveL Target_7930,v50,fine,MyNewTool\WObj:=A3;
        MoveL Target_7940,v50,fine,MyNewTool\WObj:=A3;
        MoveL Target_7950,v50,fine,MyNewTool\WObj:=A3;
        MoveL Target_7960,v50,fine,MyNewTool\WObj:=A3;
        MoveL Target_7970,v50,fine,MyNewTool\WObj:=A3;
        MoveL Target_7980,v50,fine,MyNewTool\WObj:=A3;
        MoveL Target_7990,v50,fine,MyNewTool\WObj:=A3;
        MoveL Target_8000,v50,fine,MyNewTool\WObj:=A3;
        MoveL Target_8010,v50,fine,MyNewTool\WObj:=A3;
        MoveL Target_8020,v50,fine,MyNewTool\WObj:=A3;
        MoveL Target_8030,v50,fine,MyNewTool\WObj:=A3;
        MoveL Target_8040,v50,fine,MyNewTool\WObj:=A3;
        MoveL Target_8050,v50,fine,MyNewTool\WObj:=A3;
        MoveL Target_8060,v50,fine,MyNewTool\WObj:=A3;
        MoveL Target_8070,v50,fine,MyNewTool\WObj:=A3;
        MoveL Target_8080,v50,fine,MyNewTool\WObj:=A3;
        MoveL Target_8090,v50,fine,MyNewTool\WObj:=A3;
        MoveL Target_8100,v50,fine,MyNewTool\WObj:=A3;
        MoveL Target_8110,v50,fine,MyNewTool\WObj:=A3;
        MoveL Target_8120,v50,fine,MyNewTool\WObj:=A3;
        MoveL Target_8130,v50,fine,MyNewTool\WObj:=A3;
        MoveL Target_8140,v50,fine,MyNewTool\WObj:=A3;
        MoveL Target_8150,v50,fine,MyNewTool\WObj:=A3;
        MoveL Target_8160,v50,fine,MyNewTool\WObj:=A3;
        MoveL Target_8170,v50,fine,MyNewTool\WObj:=A3;
        MoveL Target_8180,v50,fine,MyNewTool\WObj:=A3;
        MoveL Target_8190,v50,fine,MyNewTool\WObj:=A3;
        MoveL Target_8200,v50,fine,MyNewTool\WObj:=A3;
        MoveL Target_8210,v50,fine,MyNewTool\WObj:=A3;
        MoveL Target_8220,v50,fine,MyNewTool\WObj:=A3;
        MoveL Target_8230,v50,fine,MyNewTool\WObj:=A3;
        MoveL Target_8240,v50,fine,MyNewTool\WObj:=A3;
        MoveL Target_8250,v50,fine,MyNewTool\WObj:=A3;
        MoveL Target_8260,v50,fine,MyNewTool\WObj:=A3;
        MoveL Target_8270,v50,fine,MyNewTool\WObj:=A3;
        MoveL Target_8280,v50,fine,MyNewTool\WObj:=A3;
        MoveL Target_8290,v50,fine,MyNewTool\WObj:=A3;
        MoveL Target_8300,v50,fine,MyNewTool\WObj:=A3;
        MoveL Target_8310,v50,fine,MyNewTool\WObj:=A3;
        MoveL Target_8320,v50,fine,MyNewTool\WObj:=A3;
        MoveL Target_8330,v50,fine,MyNewTool\WObj:=A3;
        MoveL Target_8340,v50,fine,MyNewTool\WObj:=A3;
        MoveL Target_8350,v50,fine,MyNewTool\WObj:=A3;
        MoveL Target_8360,v50,fine,MyNewTool\WObj:=A3;
        MoveL Target_8370,v50,fine,MyNewTool\WObj:=A3;
        MoveL Target_8380,v50,fine,MyNewTool\WObj:=A3;
        MoveL Target_8390,v50,fine,MyNewTool\WObj:=A3;
        MoveL Target_8400,v50,fine,MyNewTool\WObj:=A3;
        MoveL Target_8410,v50,fine,MyNewTool\WObj:=A3;
        MoveL Target_8420,v50,fine,MyNewTool\WObj:=A3;
        MoveL Target_8430,v50,fine,MyNewTool\WObj:=A3;
        MoveL Target_8440,v50,fine,MyNewTool\WObj:=A3;
        MoveL Target_8450,v50,fine,MyNewTool\WObj:=A3;
        MoveL Target_8460,v50,fine,MyNewTool\WObj:=A3;
        MoveL Target_8470,v50,fine,MyNewTool\WObj:=A3;
        MoveL Target_8480,v50,fine,MyNewTool\WObj:=A3;
        MoveL Target_8490,v50,fine,MyNewTool\WObj:=A3;
        MoveL Target_8500,v50,fine,MyNewTool\WObj:=A3;
        MoveL Target_8510,v50,fine,MyNewTool\WObj:=A3;
        MoveL Target_8520,v50,fine,MyNewTool\WObj:=A3;
        MoveL Target_8530,v50,fine,MyNewTool\WObj:=A3;
        MoveL Target_8540,v50,fine,MyNewTool\WObj:=A3;
        MoveL Target_8550,v50,fine,MyNewTool\WObj:=A3;
        MoveL Target_8560,v50,fine,MyNewTool\WObj:=A3;
        MoveL Target_8570,v50,fine,MyNewTool\WObj:=A3;
        MoveL Target_8580,v50,fine,MyNewTool\WObj:=A3;
        MoveL Target_8590,v50,fine,MyNewTool\WObj:=A3;
        MoveL Target_8600,v50,fine,MyNewTool\WObj:=A3;
        MoveL Target_8610,v50,fine,MyNewTool\WObj:=A3;
        MoveL Target_8620,v50,fine,MyNewTool\WObj:=A3;
        MoveL Target_8630,v50,fine,MyNewTool\WObj:=A3;
        MoveL Target_8640,v50,fine,MyNewTool\WObj:=A3;
        MoveL Target_8650,v50,fine,MyNewTool\WObj:=A3;
        MoveL Target_8660,v50,fine,MyNewTool\WObj:=A3;
        MoveL Target_8670,v50,fine,MyNewTool\WObj:=A3;
        MoveL Target_8680,v50,fine,MyNewTool\WObj:=A3;
        MoveL Target_8690,v50,fine,MyNewTool\WObj:=A3;
        MoveL Target_8700,v50,fine,MyNewTool\WObj:=A3;
        MoveL Target_8710,v50,fine,MyNewTool\WObj:=A3;
        MoveL Target_8720,v50,fine,MyNewTool\WObj:=A3;
        MoveL Target_8730,v50,fine,MyNewTool\WObj:=A3;
        MoveL Target_8740,v50,fine,MyNewTool\WObj:=A3;
        MoveL Target_8750,v50,fine,MyNewTool\WObj:=A3;
        MoveL Target_8760,v50,fine,MyNewTool\WObj:=A3;
        MoveL Target_8770,v50,fine,MyNewTool\WObj:=A3;
        MoveL Target_8780,v50,fine,MyNewTool\WObj:=A3;
        MoveL Target_8790,v50,fine,MyNewTool\WObj:=A3;
        MoveL Target_8800,v50,fine,MyNewTool\WObj:=A3;
        MoveL Target_8810,v50,fine,MyNewTool\WObj:=A3;
        MoveL Target_8820,v50,fine,MyNewTool\WObj:=A3;
        MoveL Target_8830,v50,fine,MyNewTool\WObj:=A3;
        MoveL Target_8840,v50,fine,MyNewTool\WObj:=A3;
        MoveL Target_8850,v50,fine,MyNewTool\WObj:=A3;
        MoveL Target_8860,v50,fine,MyNewTool\WObj:=A3;
        MoveL Target_8870,v50,fine,MyNewTool\WObj:=A3;
        MoveL Target_8880,v50,fine,MyNewTool\WObj:=A3;
        MoveL Target_8890,v50,fine,MyNewTool\WObj:=A3;
        MoveL Target_8900,v50,fine,MyNewTool\WObj:=A3;
        MoveL Target_8910,v50,fine,MyNewTool\WObj:=A3;
        MoveL Target_8920,v50,fine,MyNewTool\WObj:=A3;
        MoveL Target_8930,v50,fine,MyNewTool\WObj:=A3;
        MoveL Target_8940,v50,fine,MyNewTool\WObj:=A3;
        MoveL Target_8950,v50,fine,MyNewTool\WObj:=A3;
        MoveL Target_8960,v50,fine,MyNewTool\WObj:=A3;
        MoveL Target_8970,v50,fine,MyNewTool\WObj:=A3;
        MoveL Target_8980,v50,fine,MyNewTool\WObj:=A3;
        MoveL Target_8990,v50,fine,MyNewTool\WObj:=A3;
        MoveL Target_9000,v50,fine,MyNewTool\WObj:=A3;
        MoveL Target_9010,v50,fine,MyNewTool\WObj:=A3;
        MoveL Target_9020,v50,fine,MyNewTool\WObj:=A3;
        MoveL Target_9030,v50,fine,MyNewTool\WObj:=A3;
        MoveL Target_9040,v50,fine,MyNewTool\WObj:=A3;
        MoveL Target_9050,v50,fine,MyNewTool\WObj:=A3;
        MoveL Target_9060,v50,fine,MyNewTool\WObj:=A3;
        MoveL Target_9070,v50,fine,MyNewTool\WObj:=A3;
        MoveL Target_9080,v50,fine,MyNewTool\WObj:=A3;
        MoveL Target_9090,v50,fine,MyNewTool\WObj:=A3;
        MoveL Target_9100,v50,fine,MyNewTool\WObj:=A3;
